# B&R Automation Studio project Assembly_and_ST (part 3)

#### Outfeed_Aborted.st
```iecst
ACTION Outfeed_Aborted:

	IF gSuperTrak.state.stateMachine.operationalState = ABORTED THEN
		//TODO: Insert Outfeed LED Light control

	ELSE
		//TODO: Insert Outfeed LED Light control
	END_IF;

	IF gSuperTrak.skill.Outfeed.state.stateMachine.stateTransition.reset THEN
		gSuperTrak.skill.Outfeed.state.stateMachine.operationalState := RESETTING;

	ELSIF gSuperTrak.skill.Outfeed.state.stateMachine.stateTransition.clear THEN
		gSuperTrak.skill.Outfeed.state.stateMachine.operationalState := CLEARING;

	END_IF;

END_ACTION
```

#### Outfeed_Stopped.st
```iecst
ACTION Outfeed_Stopped:

	IF gSuperTrak.skill.Outfeed.state.stateMachine.stateTransition.reset
	(*AND	NOT gbMessageSumAlarm*) THEN

		gSuperTrak.skill.Outfeed.state.stateMachine.operationalState := RESETTING;
	END_IF;

END_ACTION
```

#### Outfeed_Clearing.st
```iecst
ACTION Outfeed_Clearing:

	gSuperTrak.skill.Outfeed.state.stateMachine.stateTransition.clear := FALSE;

	gSuperTrak.skill.Outfeed.state.stateMachine.operationalState := STOPPED;

END_ACTION
```

#### Outfeed_Starting.st
```iecst
ACTION Outfeed_Starting:

	(* ************************************************************************** *)
	(* starting Outfeed skill *)
	IF NOT Outfeed_Full THEN
		gSuperTrak.skill.Outfeed.state.stateMachine.stateTransition.start := FALSE;
		gSuperTrak.skill.Outfeed.state.stateMachine.operationalState := RUNNING;
	END_IF;

END_ACTION
```

#### Outfeed_Completing.st
```iecst
ACTION Outfeed_Completing:
	gSuperTrak.skill.Outfeed.state.stateMachine.operationalState := COMPLETE;
END_ACTION
```

#### Outfeed_Complete.st
```iecst
ACTION Outfeed_Complete:

	Outfeed_Actuator_UP := FALSE;
	Outfeed_Actuator_DOWN := FALSE;
	Outfeed_Actuator_FRONT := FALSE;
	Outfeed_Actuator_BACK := FALSE;

	(* Skill stays in complete until trigger from MES *)
	IF gSuperTrak.skill.Outfeed.state.stateMachine.stateTransition.reset THEN
		gSuperTrak.skill.Outfeed.state.stateMachine.operationalState := RESETTING;
	END_IF;

END_ACTION
```

#### Outfeed_Holding.st
```iecst
ACTION Outfeed_Holding:

	gSuperTrak.skill.Outfeed.state.stateMachine.operationalState := HELD;

END_ACTION
```

#### Outfeed_Suspended.st
```iecst
ACTION Outfeed_Suspended:

	IF gSuperTrak.skill.Outfeed.state.stateMachine.stateTransition.unsuspend THEN
		gSuperTrak.skill.Outfeed.state.stateMachine.operationalState := UNSUSPENDING;
	END_IF;

END_ACTION
```

#### Outfeed_Unsuspending.st
```iecst
ACTION Outfeed_Unsuspending:

	gSuperTrak.skill.Outfeed.state.stateMachine.operationalState := RUNNING;

END_ACTION
```

#### Outfeed_Running.st
```iecst
ACTION Outfeed_Running:

	IF NOT Outfeed_Full AND Outfeed_Checked THEN
		(*Activate actuator movement up and wait until fully extended*)

		Outfeed_Actuator_UP := TRUE;

		Timer_Outfeed_UP(IN := TRUE, PT := T#10s);

		IF Timer_Outfeed_UP.Q THEN
			Outfeed_LED_Green := TRUE;
			Outfeed_LED_Red := FALSE;
			Outfeed_LED_Blue := FALSE;

			Outfeed_Actuator_FRONT := TRUE;
			Timer_Outfeed_FRONT(IN:= TRUE, PT:=T#5s);

			IF Timer_Outfeed_FRONT.Q THEN

				(*Actuator go down and then we get complete*)
				Outfeed_Actuator_UP := FALSE;
				Outfeed_Actuator_FRONT := FALSE;

				IF NOT Outfeed_Actuator_UP AND NOT Outfeed_Actuator_FRONT THEN
					Outfeed_Actuator_DOWN := TRUE;
					Outfeed_Actuator_BACK := TRUE;
				END_IF;

				Timer_Outfeed_DOWN(IN := Outfeed_Actuator_DOWN, PT := T#10s);
				Timer_Outfeed_BACK(IN := Outfeed_Actuator_BACK, PT := T#5s);

				IF Timer_Outfeed_DOWN.Q AND Timer_Outfeed_BACK.Q THEN
					Timer_Outfeed_DOWN(IN := FALSE);
					Timer_Outfeed_BACK(IN := FALSE);
					Timer_Outfeed_FRONT(IN := FALSE);
					Timer_Outfeed_UP (IN := FALSE);
					gSuperTrak.skill.Outfeed.state.stateMachine.operationalState := COMPLETING;
				END_IF;

			END_IF;

		END_IF;

	ELSIF NOT Outfeed_Checked THEN

		IF Outfeed_Full THEN
			Event_Code := 80;
			EventLog.Commands.WriteUserEvent := TRUE;

		ELSE
			Outfeed_Checked := TRUE;
		END_IF;

	END_IF;

END_ACTION
```

#### QACheck.st
```iecst
ACTION QACheck:
		(*************************************************************************************************)
		(*************************************************************************************************)
		(* State Machine *)
	CASE gSuperTrak.skill.QACheck.state.stateMachine.operationalState OF
		(*************************************************************************************************)
		(* RESETTING *)
		RESETTING:
			(*gSuperTrak.skill.QACheck.state.stateMachine.stateTransition.reset := FALSE;*)

			IF gSuperTrak.skill.QACheck.state.stateMachine.stateTransition.abort THEN
				gSuperTrak.skill.QACheck.state.stateMachine.operationalState := ABORTING;

			ELSIF gSuperTrak.skill.QACheck.state.stateMachine.stateTransition.stop THEN
				gSuperTrak.skill.QACheck.state.stateMachine.operationalState := STOPPING;

			ELSE
				QACheck_Resetting;

			END_IF;

		(*************************************************************************************************)
		(* IDLE *)
		IDLE:
			gSuperTrak.skill.QACheck.state.stateMachine.stateTransition.reset := FALSE;

			IF gSuperTrak.skill.QACheck.state.stateMachine.stateTransition.abort THEN
				gSuperTrak.skill.QACheck.state.stateMachine.operationalState := ABORTING;

			ELSIF gSuperTrak.skill.QACheck.state.stateMachine.stateTransition.stop THEN
				gSuperTrak.skill.QACheck.state.stateMachine.operationalState := STOPPING;

			ELSE
				QACheck_Idle;

			END_IF;

		(*************************************************************************************************)
		(* STARTING *)
		STARTING:
//			gSuperTrak.skill.QACheck.state.stateMachine.stateTransition.start := FALSE;

			IF gSuperTrak.skill.QACheck.state.stateMachine.stateTransition.abort THEN
				gSuperTrak.skill.QACheck.state.stateMachine.operationalState := ABORTING;

			ELSIF gSuperTrak.skill.QACheck.state.stateMachine.stateTransition.stop THEN
				gSuperTrak.skill.QACheck.state.stateMachine.operationalState := STOPPING;

			ELSE
				QACheck_Starting;

			END_IF;

		(*************************************************************************************************)
		(* RUNNING *)
		RUNNING:

			gSuperTrak.skill.QACheck.state.stateMachine.stateTransition.start := FALSE;

			IF gSuperTrak.skill.QACheck.state.stateMachine.stateTransition.abort THEN
				gSuperTrak.skill.QACheck.state.stateMachine.operationalState := ABORTING;

			ELSIF gSuperTrak.skill.QACheck.state.stateMachine.stateTransition.stop THEN
				gSuperTrak.skill.QACheck.state.stateMachine.operationalState := STOPPING;

			ELSIF gSuperTrak.skill.QACheck.state.stateMachine.stateTransition.hold THEN

				//				gSuperTrak.skill.QACheck.state.stateMachine.operationalState := HOLDING;

			ELSIF gSuperTrak.skill.QACheck.state.stateMachine.stateTransition.suspend THEN

				//				gSuperTrak.skill.QACheck.state.stateMachine.operationalState := SUSPENDING;

			ELSIF gSuperTrak.skill.QACheck.state.stateMachine.stateTransition.pause THEN

				//				gSuperTrak.skill.QACheck.state.stateMachine.operationalState := PAUSING;

			ELSE
				QACheck_Running;

			END_IF;

		(*************************************************************************************************)
		(* PAUSING *)
		PAUSING:
			(*gSuperTrak.skill.QACheck.state.stateMachine.stateTransition.pause := FALSE;*)

			IF gSuperTrak.skill.QACheck.state.stateMachine.stateTransition.abort THEN
				gSuperTrak.skill.QACheck.state.stateMachine.operationalState := ABORTING;

			ELSIF gSuperTrak.skill.QACheck.state.stateMachine.stateTransition.stop THEN
				gSuperTrak.skill.QACheck.state.stateMachine.operationalState := STOPPING;

			ELSIF gSuperTrak.skill.QACheck.state.stateMachine.stateTransition.hold THEN

				//				gSuperTrak.skill.QACheck.state.stateMachine.operationalState := HOLDING;

			ELSIF gSuperTrak.skill.QACheck.state.stateMachine.stateTransition.suspend THEN

				//				gSuperTrak.skill.QACheck.state.stateMachine.operationalState := SUSPENDING;

			ELSE
				QACheck_Pausing;
			END_IF;

		(*************************************************************************************************)
		(* PAUSED *)
		PAUSED:

			gSuperTrak.skill.QACheck.state.stateMachine.stateTransition.pause := FALSE;

			IF gSuperTrak.skill.QACheck.state.stateMachine.stateTransition.abort THEN
				gSuperTrak.skill.QACheck.state.stateMachine.operationalState := ABORTING;

			ELSIF gSuperTrak.skill.QACheck.state.stateMachine.stateTransition.stop THEN
				gSuperTrak.skill.QACheck.state.stateMachine.operationalState := STOPPING;

			ELSIF gSuperTrak.skill.QACheck.state.stateMachine.stateTransition.hold THEN

				//				gSuperTrak.skill.QACheck.state.stateMachine.operationalState := HOLDING;

			ELSIF gSuperTrak.skill.QACheck.state.stateMachine.stateTransition.suspend THEN

				//				gSuperTrak.skill.QACheck.state.stateMachine.operationalState := SUSPENDING;

			ELSE
				QACheck_Paused;

			END_IF;

		(*************************************************************************************************)
		(* SUSPENDING *)
		SUSPENDING:
			(*gSuperTrak.skill.QACheck.state.stateMachine.stateTransition.suspend := FALSE;*)

			IF gSuperTrak.skill.QACheck.state.stateMachine.stateTransition.abort THEN
				gSuperTrak.skill.QACheck.state.stateMachine.operationalState := ABORTING;

			ELSIF gSuperTrak.skill.QACheck.state.stateMachine.stateTransition.stop THEN
				gSuperTrak.skill.QACheck.state.stateMachine.operationalState := STOPPING;

			ELSIF gSuperTrak.skill.QACheck.state.stateMachine.stateTransition.hold THEN

				//				gSuperTrak.skill.QACheck.state.stateMachine.operationalState := HOLDING;

			ELSE
				QACheck_Suspending;

			END_IF;

		(*************************************************************************************************)
		(* SUSPENDED *)
		SUSPENDED:

			gSuperTrak.skill.QACheck.state.stateMachine.stateTransition.suspend := FALSE;

			IF gSuperTrak.skill.QACheck.state.stateMachine.stateTransition.abort THEN
				gSuperTrak.skill.QACheck.state.stateMachine.operationalState := ABORTING;

			ELSIF gSuperTrak.skill.QACheck.state.stateMachine.stateTransition.stop THEN
				gSuperTrak.skill.QACheck.state.stateMachine.operationalState := STOPPING;

			ELSIF gSuperTrak.skill.QACheck.state.stateMachine.stateTransition.hold THEN

				//				gSuperTrak.skill.QACheck.state.stateMachine.operationalState := HOLDING;

			ELSE
				QACheck_Suspended;

			END_IF;

		(*************************************************************************************************)
		(* UNSUSPENDING *)
		UNSUSPENDING:
			gSuperTrak.skill.QACheck.state.stateMachine.stateTransition.unsuspend := FALSE;

			IF gSuperTrak.skill.QACheck.state.stateMachine.stateTransition.abort THEN
				gSuperTrak.skill.QACheck.state.stateMachine.operationalState := ABORTING;

			ELSIF gSuperTrak.skill.QACheck.state.stateMachine.stateTransition.stop THEN
				gSuperTrak.skill.QACheck.state.stateMachine.operationalState := STOPPING;

			ELSIF gSuperTrak.skill.QACheck.state.stateMachine.stateTransition.hold THEN

				//				gSuperTrak.skill.QACheck.state.stateMachine.operationalState := HOLDING;

			ELSE
				QACheck_Unsuspending;

			END_IF;

		(*************************************************************************************************)
		(* HOLDING *)
		HOLDING:
			(*gSuperTrak.skill.QACheck.state.stateMachine.stateTransition.hold := FALSE;*)

			IF gSuperTrak.skill.QACheck.state.stateMachine.stateTransition.abort THEN
				gSuperTrak.skill.QACheck.state.stateMachine.operationalState := ABORTING;

			ELSIF gSuperTrak.skill.QACheck.state.stateMachine.stateTransition.stop THEN
				gSuperTrak.skill.QACheck.state.stateMachine.operationalState := STOPPING;

			ELSE
				QACheck_Holding;

			END_IF;

		(*************************************************************************************************)
		(* HELD *)
		HELD:

			gSuperTrak.skill.QACheck.state.stateMachine.stateTransition.hold := FALSE;

			IF gSuperTrak.skill.QACheck.state.stateMachine.stateTransition.abort THEN
				gSuperTrak.skill.QACheck.state.stateMachine.operationalState := ABORTING;

			ELSIF gSuperTrak.skill.QACheck.state.stateMachine.stateTransition.stop THEN
				gSuperTrak.skill.QACheck.state.stateMachine.operationalState := STOPPING;

			ELSE
				QACheck_Held;

			END_IF;

		(*************************************************************************************************)
		(* UNHOLDING *)
		UNHOLDING:
			gSuperTrak.skill.QACheck.state.stateMachine.stateTransition.unhold := FALSE;

			IF gSuperTrak.skill.QACheck.state.stateMachine.stateTransition.abort THEN
				gSuperTrak.skill.QACheck.state.stateMachine.operationalState := ABORTING;

			ELSIF gSuperTrak.skill.QACheck.state.stateMachine.stateTransition.stop THEN
				gSuperTrak.skill.QACheck.state.stateMachine.operationalState := STOPPING;

			ELSE
				QACheck_Unholding;

			END_IF;

		(*************************************************************************************************)
		(* COMPLETING *)
		COMPLETING:

			IF gSuperTrak.skill.QACheck.state.stateMachine.stateTransition.abort THEN
				gSuperTrak.skill.QACheck.state.stateMachine.operationalState := ABORTING;

			ELSIF gSuperTrak.skill.QACheck.state.stateMachine.stateTransition.stop THEN
				gSuperTrak.skill.QACheck.state.stateMachine.operationalState := STOPPING;

			ELSE
				QACheck_Completing;

			END_IF;

		(*************************************************************************************************)
		(* COMPLETE *)
		COMPLETE:

			IF gSuperTrak.skill.QACheck.state.stateMachine.stateTransition.abort THEN
				gSuperTrak.skill.QACheck.state.stateMachine.operationalState := ABORTING;

			ELSIF gSuperTrak.skill.QACheck.state.stateMachine.stateTransition.stop THEN
				gSuperTrak.skill.QACheck.state.stateMachine.operationalState := STOPPING;

			ELSE
				QACheck_Complete;

			END_IF;

		(*************************************************************************************************)
		(* STOPPING *)
		STOPPING:
//			gSuperTrak.skill.QACheck.state.stateMachine.stateTransition.stop := FALSE;

			IF gSuperTrak.skill.QACheck.state.stateMachine.stateTransition.abort THEN
				gSuperTrak.skill.QACheck.state.stateMachine.operationalState := ABORTING;

			ELSE
				QACheck_Stopping;

			END_IF;

		(*************************************************************************************************)
		(* STOPPED *)
		STOPPED:

			gSuperTrak.skill.QACheck.state.stateMachine.stateTransition.stop := FALSE;

			IF gSuperTrak.skill.QACheck.state.stateMachine.stateTransition.abort THEN
				gSuperTrak.skill.QACheck.state.stateMachine.operationalState := ABORTING;

			ELSE
				QACheck_Stopped;

			END_IF;

		(*************************************************************************************************)
		(* ABORTING *)
		ABORTING:
			(*gSuperTrak.skill.QACheck.state.stateMachine.stateTransition.abort := FALSE;*)

			QACheck_Aborting;

		(*************************************************************************************************)
		(* ABORTED *)
		ABORTED:

			gSuperTrak.skill.QACheck.state.stateMachine.stateTransition.abort := FALSE;

			QACheck_Aborted;

		(*************************************************************************************************)
		(* CLEARING *)
		CLEARING:
			gSuperTrak.skill.QACheck.state.stateMachine.stateTransition.clear := FALSE;

			QACheck_Clearing;

			(*************************************************************************************************)
			(* ELSE *)
		ELSE;

	END_CASE;
END_ACTION
```

#### QACheck_Aborting.st
```iecst
ACTION QACheck_Aborting:

//	IF NOT Transition_From_Stopped AND gSuperTrak.state.stateMachine.operationalState <> ABORTING THEN
//		Event_Code := 77;
//		EventLog.Commands.WriteUserEvent := TRUE;
//	END_IF;
//

	//Not knowing if any trigger was set to true before the abort we make sure every one of them is false before going to aborted
	gSuperTrak.skill.QACheck.state.stateMachine.stateTransition.abort 		:= FALSE;
	gSuperTrak.skill.QACheck.state.stateMachine.stateTransition.clear 		:= FALSE;
	gSuperTrak.skill.QACheck.state.stateMachine.stateTransition.hold 		:= FALSE;
	gSuperTrak.skill.QACheck.state.stateMachine.stateTransition.pause 		:= FALSE;
	gSuperTrak.skill.QACheck.state.stateMachine.stateTransition.reset 		:= FALSE;
	gSuperTrak.skill.QACheck.state.stateMachine.stateTransition.resume 		:= FALSE;
	gSuperTrak.skill.QACheck.state.stateMachine.stateTransition.start 		:= FALSE;
	gSuperTrak.skill.QACheck.state.stateMachine.stateTransition.stop 		:= FALSE;
	gSuperTrak.skill.QACheck.state.stateMachine.stateTransition.suspend 	:= FALSE;
	gSuperTrak.skill.QACheck.state.stateMachine.stateTransition.unhold 		:= FALSE;
	gSuperTrak.skill.QACheck.state.stateMachine.stateTransition.unsuspend 	:= FALSE;

	LED_Red   := TRUE;
	LED_Green := FALSE;
	LED_Blue  := FALSE;
	QA_Actuator_UP := FALSE;

	QA_Actuator_DOWN := FALSE;

	Skills_Aborted := Skills_Aborted + 1;
	gSuperTrak.skill.QACheck.state.stateMachine.operationalState := ABORTED;

END_ACTION
```

#### QACheck_Aborted.st
```iecst
ACTION QACheck_Aborted:

	IF gSuperTrak.state.stateMachine.operationalState = ABORTED THEN
		LED_Blue := TRUE;
		LED_Green := FALSE;
		LED_Red := FALSE;

	ELSE
		LED_Blue := FALSE;
		LED_Green := FALSE;
		LED_Red := TRUE;
	END_IF;

	IF gSuperTrak.skill.QACheck.state.stateMachine.stateTransition.reset THEN
		gSuperTrak.skill.QACheck.state.stateMachine.operationalState := RESETTING;

	ELSIF gSuperTrak.skill.QACheck.state.stateMachine.stateTransition.clear THEN
		gSuperTrak.skill.QACheck.state.stateMachine.operationalState := CLEARING;

	END_IF;

END_ACTION
```

#### QACheck_Clearing.st
```iecst
ACTION QACheck_Clearing:

	gSuperTrak.skill.QACheck.state.stateMachine.stateTransition.clear := FALSE;

	gSuperTrak.skill.QACheck.state.stateMachine.operationalState := STOPPED;

END_ACTION
```

#### QACheck_Idle.st
```iecst
ACTION QACheck_Idle:

	LED_Green := FALSE;
	LED_Red := FALSE;
	LED_Blue := TRUE;

	IF gSuperTrak.skill.QACheck.state.stateMachine.stateTransition.start THEN

		gSuperTrak.skill.QACheck.state.stateMachine.operationalState := STARTING;

	END_IF

	QA_Actuator_UP := FALSE;
	QA_Actuator_DOWN := FALSE;

END_ACTION
```

#### QACheck_Starting.st
```iecst
ACTION QACheck_Starting:

	(* ************************************************************************** *)
	(* starting QACheck skill *)
	gSuperTrak.skill.QACheck.state.stateMachine.stateTransition.start := FALSE;
	gSuperTrak.skill.QACheck.state.stateMachine.operationalState := RUNNING;

END_ACTION
```

#### QACheck_Completing.st
```iecst
ACTION QACheck_Completing:

	(* Alarms Handling?? *)

	(*Actuator go down and then we get complete*)
	QA_Actuator_UP := FALSE;
	LED_Green := FALSE;
	LED_Red := TRUE;
	LED_Blue := FALSE;
	Timer_Enable_Barrier(IN := LED_Red, PT := T#0.5s);

	IF Timer_Enable_Barrier.Q THEN
		Disable_Light_Barrier := FALSE;
	END_IF;

	IF NOT QA_Actuator_UP THEN
		QA_Actuator_DOWN := TRUE;
	END_IF;

	Timer_Actuator_DOWN(IN := QA_Actuator_DOWN, PT := T#8s);

	IF Timer_Actuator_DOWN.Q AND NOT Disable_Light_Barrier THEN
		gSuperTrak.skill.QACheck.state.stateMachine.operationalState := COMPLETE;
		Timer_Actuator_DOWN(IN := FALSE);
	END_IF;

END_ACTION
```

#### QACheck_Complete.st
```iecst
ACTION QACheck_Complete:
	(* Skill stays in complete until trigger from MES *)
	IF gSuperTrak.skill.QACheck.state.stateMachine.stateTransition.reset THEN
		gSuperTrak.skill.QACheck.state.stateMachine.operationalState := RESETTING;
	END_IF;

	Timer_Enable_Barrier(IN := FALSE);
	QA_Actuator_UP := FALSE;
	QA_Actuator_DOWN := FALSE;

END_ACTION
```

#### QACheck_Running.st
```iecst
ACTION QACheck_Running:
	(*Activate actuator movement up and wait until fully extended*)

	Timer_Actuator_UP(IN := QA_Actuator_UP, PT := T#8s);
	QA_Actuator_UP := TRUE;

	IF Timer_Actuator_UP.Q THEN
		LED_Green := TRUE;
		LED_Red := FALSE;
		LED_Blue := FALSE;
		Disable_Light_Barrier := TRUE;
	END_IF;

	IF QA_finished THEN
		QA_finished := FALSE;
		QA_Actuator_UP := FALSE;
		Timer_Actuator_UP(IN := FALSE);
		gSuperTrak.skill.QACheck.state.stateMachine.operationalState := COMPLETING;
	END_IF;

END_ACTION
```

### UsrEventHandling.typ
```iecst
(*******************************************************************
 * Local data types of program EventLog
 ********************************************************************)

TYPE
	EventLog_typ : 	STRUCT  (*Event handling.*)
		Commands : EventLog_Commands_typ; (*Event handling user commands.*)
		Data : EventLog_Data_typ; (*Event handling data for state machine.*)
		Event : EventLog_Event_typ; (*Event handling event description.*)
		FunctionBlocks : EventLog_FunctionBlocks_typ; (*Event handling used function blocks.*)
	END_STRUCT;
	EventLog_Data_typ : 	STRUCT
		Step : EventLogSteps; (*Current step. STEP_ERROR must be manually reset (STEP_WAIT_FOR_INPUT).*)
		Ident : ArEventLogIdentType; (*Ident of the logbook "UsrEvLog".*)
		StatusID : DINT; (*Status information for STEP_ERROR.*)
		GetIdentOkNextStep : EventLogSteps; (*Internal helper for state machine.*)
		GetIdentFailNextStep : EventLogSteps; (*Internal helper for state machine.*)
	END_STRUCT;
	EventLog_Event_typ : 	STRUCT
		Severity : USINT; (*Severity of the last event (read).*)
		Customer : BOOL; (*Customer bit of the last event (read).*)
		Facility : UINT; (*Facility of the last event (read).*)
		Code : UINT; (*Code of the last event (read).*)
		EventID : DINT; (*EventID for write event (write - is not set by reading an event).*)
		ErrorNumber : UDINT; (*Error number of the event - set when the read event is no event id event (read).*)
		EnteredBy : STRING[36]; (*User/object identification (read/write - optional).*)
		OriginID : ArEventLogRecordIDType; (*Record id of the origin record (read/write - optional).*)
		RecordID : ArEventLogRecordIDType; (*Record id of the event to read (read - set automatically).*)
		TimeStamp : ArEventLogTimeStampType;
		AdditionalDataSize : UDINT; (*Size of the additional data (read/write - optional)*)
		AdditionalDataFormat : USINT; (*Format of the additional data (read/write)*)
		AdditionalData : STRING[255]; (*Additional data (read/write)*)
	END_STRUCT;
	EventLog_FunctionBlocks_typ : 	STRUCT
		ArEventLogCreate_0 : ArEventLogCreate;
		ArEventLogDelete_0 : ArEventLogDelete;
		ArEventLogGetIdent_0 : ArEventLogGetIdent;
		ArEventLogGetLatestRecordID_0 : ArEventLogGetLatestRecordID;
		ArEventLogGetPreviousRecordID_0 : ArEventLogGetPreviousRecordID;
		ArEventLogWrite_0 : ArEventLogWrite;
		ArEventLogRead_0 : ArEventLogRead;
		ArEventLogReadErrorNumber_0 : ArEventLogReadErrorNumber;
		ArEventLogReadAddData_0 : ArEventLogReadAddData;
		ArEventLogReadObjectID_0 : ArEventLogReadObjectID;
	END_STRUCT;
	EventLogSteps :
		(
		STEP_WAIT_FOR_INPUT := 0,
		STEP_CREATE_LOGBOOK := 1,
		STEP_DELETE_LOGBOOK := 2,
		STEP_GET_LOGBOOK_IDENT := 3,
		STEP_WRITE_EVENT := 4,
		STEP_READ_EVENT := 5,
		STEP_READ_ERROR_NUMBER := 6,
		STEP_READ_ADDITIONAL_DATA := 7,
		STEP_READ_OBJECT_ID := 8,
		STEP_GET_LATEST_RECORD_ID := 9,
		STEP_GET_PREVIOUS_RECORD_ID := 10,
		STEP_ERROR := 255
		);
END_TYPE

(*
Copyright ATS Automation Tooling Systems, Inc. 2015-2016
All rights reserved.
*)
(********************************************************************
 * COPYRIGHT --
 ********************************************************************
 * File: Global.typ
 * Author: VM_User
 * Created: 14. März 2014
 ********************************************************************
 * Global data types of project T1
 ********************************************************************)
(***********************************************************************)
(*Variables for Event logger control and definition*)
(**********************************************************************)

TYPE
	EventLog_Commands_typ : 	STRUCT
		CreateUserLog : BOOL; (*Creates the user logbook "UsrEvLog" in USERROM.*)
		DeleteUserLog : BOOL; (*Deletes the user logbook "UsrEvLog".*)
		WriteUserEvent : BOOL; (*Writes a user event into the user logbook "UsrEvLog". *)
		ReadLatestEvent : BOOL; (*Reads the latest event of the user logbook "UsrEvLog".*)
		ReadPreviousEvent : BOOL; (*Reads the previous event (of the given record id) of the user logbook "UserEvLog".*)
	END_STRUCT;
	Event_Codes_Typ : 	STRUCT
		Severity_Code : USINT;
		Facility_Code : USINT;
		Code_Value : USINT;
		ID : DINT;
		Event_Message : STRING[256]; (*Message for the event generated*)
	END_STRUCT;
END_TYPE
```

### UsrEventHandling.var
```iecst
(* ============================================================
Variable for known events definition
   ============================================================ *)
VAR
	Events : ARRAY[0..250] OF Event_Codes_Typ;
	Event_Code : UINT;
END_VAR
(*******************************************************************
 * Variables of program EventLog
 ********************************************************************)
VAR
	EventLog : EventLog_typ; (*Event handling.*)
END_VAR
(*=============================================================*)
(*Variables for info events writing control*)
(*=============================================================*)
VAR
	Write_Info : BOOL;
	ST_Last_Info_Written : UINT;
	Assembly_Last_Info_Written : UINT;
	General_Last_Info_Written : UINT;
	Last_Event_Written : UINT;
	Set_Info_Messages : BOOL;
	Restart_Status : UINT;
	Initialization : BOOL;
END_VAR
(*=============================================================*)
(*Flags for new events *)
(*=============================================================*)
VAR
	Info_Event : BOOL;
	New_Event : BOOL;
END_VAR
(********************************************************************************************)
(* Variables for Error Detection *)
(********************************************************************************************)
VAR
	SumCritical : BOOL;
END_VAR
```

### Program Logical/Events_handling/AlarmHandling

#### Variables.var
```iecst
VAR
	i : USINT;
	iEvent : USINT := 0;
END_VAR
(********************************************************************************************)
(* Variables for Service Stations *)
(********************************************************************************************)
VAR
END_VAR
```

#### Main.st
```iecst
PROGRAM _INIT
	(*Initial definiton of all the messages that could possibly be used during the execution*)
	ST_Events_Data;
	Assembly_Events_Data;
	General_Events_Data;

	(*Flag for the user to select whether or not the info messages of the actual state of the state machines will be shown*)
	//By default is false taking into account that if not this could generate execesive information in the logger
	Set_Info_Messages := FALSE;
	SumCritical := FALSE;

	Initialization := TRUE;

END_PROGRAM

PROGRAM _CYCLIC
	ComauerrorHandler;
	STerrorHandler;
	RefillEvent;
	ErrorSum;
	(* Error Reset *)

	IF gSuperTrak.state.errorAcknowledge AND SumCritical THEN

		IF Last_Event_Written = 200  AND NOT Initialization THEN
			Event_Code := 201;
			EventLog.Commands.WriteUserEvent := TRUE;

			Restart_Status := SYSreset(1, 1); (* perform WARMSTART *)

			IF Restart_Status <> 0 THEN (* check status value *)
				Event_Code := 202;
				EventLog.Commands.WriteUserEvent := TRUE;
			END_IF;

		END_IF;

		Event_Code := 249;
		EventLog.Commands.WriteUserEvent := TRUE;
		Initialization := FALSE;

		gSuperTrak.state.errorAcknowledge := FALSE;
		SumCritical := FALSE;

	END_IF;

	IF gAssemblyModule.state.errorAcknowledge AND SumCritical THEN

		IF Last_Event_Written = 200  AND NOT Initialization THEN
			Event_Code := 201;
			EventLog.Commands.WriteUserEvent := TRUE;

			Restart_Status := SYSreset(1, 1); (* perform WARMSTART *)

			IF Restart_Status <> 0 THEN (* check status value *)
				Event_Code := 202;
				EventLog.Commands.WriteUserEvent := TRUE;
			END_IF;

		END_IF;

		Event_Code := 249;
		EventLog.Commands.WriteUserEvent := TRUE;

		gAssemblyModule.state.errorAcknowledge := FALSE;
		SumCritical := FALSE;

	END_IF;

	StateInfo;
	ServiceStations;
	Assembly_WarningHandler;

	(* Call to the skills responsible of the critical errors detection and duplicate messages management*)
	IF New_Event THEN
		InfoHistory;
	END_IF;

END_PROGRAM
```

#### ComauErrorHandler.st
```iecst
ACTION ComauerrorHandler:

	IF Event_Code = 101 THEN

		Mp_Comau.ErrorReset := TRUE;

		Plastic_Cup_Supply_Position[0] := PLASTIC_CUP_INIT_POSITION [0];
		Plastic_Cup_Supply_Position[1] := PLASTIC_CUP_INIT_POSITION [1];
		Plastic_Cup_Supply_Position[2] := PLASTIC_CUP_INIT_POSITION [2];

		Plastic_Cup_Supply_Above_Pos[0] := PLASTIC_CUP_INIT_POSITION [0];
		Plastic_Cup_Supply_Above_Pos[1] := PLASTIC_CUP_INIT_POSITION [1];
		Plastic_Cup_Supply_Above_Pos[2] := PLASTIC_CUP_INIT_POSITION [2] + 60;

		x_counter_plastic := 0;
		y_counter_plastic := 0;

		Paper_Cup_Supply_Position[0] := PAPER_CUP_INIT_POSITION [0];
		Paper_Cup_Supply_Position[1] := PAPER_CUP_INIT_POSITION [1];
		Paper_Cup_Supply_Position[2] := PAPER_CUP_INIT_POSITION [2];

		Paper_Cup_Supply_Above_Pos[0] := PAPER_CUP_INIT_POSITION [0];
		Paper_Cup_Supply_Above_Pos[1] := PAPER_CUP_INIT_POSITION [1];
		Paper_Cup_Supply_Above_Pos[2] := PAPER_CUP_INIT_POSITION [2] + 60;

		x_counter_plastic := 0;
		y_counter_plastic := 0;

		IF NOT Mp_Comau.Error THEN
			Mp_Comau.ErrorReset := FALSE;
		END_IF;

	END_IF;

	IF Event_Code = 102 THEN  //Error in imput parameter paper cup
		gAssemblyModule.skill.provideCup.inputParameters.cupType :=0;
	END_IF;

	IF Event_Code = 131 //Error In Homing Procedure
		OR Event_Code = 100 THEN //Clearing Timeout

		Mp_Comau.ErrorReset := TRUE;
		Mp_Comau.Home := FALSE;
		HomeRobot := FALSE;

		IF NOT Mp_Comau.Error THEN
			Mp_Comau.ErrorReset := FALSE;
		END_IF;

	END_IF;

END_ACTION
```

#### STErrorHandler.st
```iecst
ACTION STerrorHandler:

	IF StControl_0.Error THEN
		Event_Code := 1;
		EventLog.Commands.WriteUserEvent := TRUE;
	END_IF;

END_ACTION
```

#### ErrorAcknowledgement.st - not listed in the package file held
```iecst
ACTION ErrorAcknowledgement:
	(* Error Reset *)
	IF gSuperTrak.state.errorAcknowledge AND SumCritical THEN

		Event_Code := 249;
		EventLog.Commands.WriteUserEvent := TRUE;

		gSuperTrak.state.errorAcknowledge := FALSE;
		SumCritical := FALSE;

	END_IF;

	IF gAssemblyModule.state.errorAcknowledge AND SumCritical THEN

		Event_Code := 249;
		EventLog.Commands.WriteUserEvent := TRUE;

		gAssemblyModule.state.errorAcknowledge := FALSE;
		SumCritical := FALSE;
	END_IF;

END_ACTION
```

#### InfoHistory.st
```iecst
ACTION InfoHistory:

	EventLog.Commands.ReadLatestEvent := TRUE;

	IF EventLog.FunctionBlocks.ArEventLogReadObjectID_0.Done THEN

		IF Info_Event THEN

			IF EventLog.Event.Code < 100 THEN
				ST_Last_Info_Written := EventLog.Event.Code;

			ELSIF EventLog.Event.Code < 200 THEN
				Assembly_Last_Info_Written := EventLog.Event.Code;

			ELSE
				General_Last_Info_Written := EventLog.Event.Code;
			END_IF;

		ELSE

			Last_Event_Written := EventLog.Event.Code;

		END_IF;

		New_Event := FALSE;

	END_IF;

END_ACTION
```

#### Refill_Event.st
```iecst
ACTION RefillEvent:

	//If a refill event is reached the module will be held, as well as the skill that detected the empty storage
	IF Event_Code = 130 THEN

		Assem_IgnoreSafetySensors := TRUE;

		IF Assem_PaperRemaining = 0 THEN
			Paper_RefillDone := FALSE;
		END_IF;

		IF Assem_PlasticRemaining = 0 THEN
			Plastic_RefillDone := FALSE;
		END_IF;

		IF gAssemblyModule.skill.provideCup.state.stateMachine.operationalState = RUNNING THEN

			gAssemblyModule.skill.provideCup.state.stateMachine.stateTransition.hold := TRUE;

		END_IF;

		IF gAssemblyModule.skill.providePellet.state.stateMachine.operationalState = RUNNING THEN

			gAssemblyModule.skill.providePellet.state.stateMachine.stateTransition.hold := TRUE;

		END_IF;

		gAssemblyModule.state.stateMachine.stateTransition.hold := TRUE;

	END_IF;

	//If a refill event is reached the module will be held, as well as the skill that detected the empty storage
	IF Event_Code = 133 THEN

		IF gAssemblyModule.skill.provideCup.state.stateMachine.operationalState = HELD THEN

			gAssemblyModule.skill.provideCup.state.stateMachine.stateTransition.unhold := TRUE;

		END_IF;

		IF gAssemblyModule.skill.providePellet.state.stateMachine.operationalState = HELD THEN

			gAssemblyModule.skill.providePellet.state.stateMachine.stateTransition.unhold := TRUE;

		END_IF;

		gAssemblyModule.state.stateMachine.stateTransition.unhold := TRUE;

	END_IF;

	IF Last_Event_Written = 133 THEN
		Event_Code := 141;
		EventLog.Commands.WriteUserEvent := TRUE;
	END_IF;

	IF gAssemblyModule.state.stateMachine.operationalState = RUNNING THEN

		//Assem_IgnoreSafetySensors := FALSE;
		gAssemblyModule.state.stateMachine.stateTransition.unhold := FALSE;

	END_IF;

	//When the refill has been completed the three refill variables will be true and the pellets will be
	//detected by the light barrier
	IF Plastic_RefillDone AND Paper_RefillDone AND Assem_PelletPresent THEN
		Refill_Done := TRUE;
	END_IF;

END_ACTION
```

#### Demo_Mode.st - not listed in the package file held
```iecst
ACTION Demo_Mode:
//Mode where the whole process can be simulated wothout needing an MES execution.
//Only SuperTrak is controlled and the modules interaction is faked using timers for a realistic execution.

	IF gSuperTrak.state.stateMachine.operationalState = ABORTED
		AND SumCritical = FALSE THEN

		gSuperTrak.state.stateMachine.stateTransition.clear := TRUE;

	END_IF;

	IF gSuperTrak.state.stateMachine.operationalState = STOPPED THEN

		gSuperTrak.state.stateMachine.stateTransition.reset := TRUE;

	END_IF;

	IF gSuperTrak.state.stateMachine.operationalState = IDLE THEN

		gSuperTrak.state.stateMachine.stateTransition.start := TRUE;

	END_IF;

	IF  gSuperTrak.state.stateMachine.operationalState = RUNNING AND
		Place_Order AND (ID = 0 OR ID = -1) THEN

		//Call skill checkParking to retrieve shuttleID

		gSuperTrak.skill.checkParking.state.stateMachine.stateTransition.start := TRUE;

		//When skill is finished store the ID in a variable
		IF gSuperTrak.skill.checkParking.state.stateMachine.operationalState = COMPLETE THEN

			ID := gSuperTrak.skill.checkParking.outputParameters.shuttleId;
			gSuperTrak.skill.checkParking.state.stateMachine.stateTransition.reset := TRUE;

		END_IF;

	END_IF;

	//checkParking returns -1 if there is no shuttle there at the station
	IF ID <> -1 AND ID <> 0 AND StTargetExt_[1].PalletPresent THEN

		Place_Order := FALSE;
		ID := 0;
		TargetControlParameters[1].AdvancedReleaseConfig.DestinationTarget := 2;
		StTargetExt_[1].ReleaseToTarget := TRUE;

		IF EDGENEG(StTargetExt_[1].PalletPresent) THEN

			StTargetExt_[1].ReleaseToTarget := FALSE;

		END_IF;

	END_IF;

	//Assembly Module
	IF StTargetExt_[2].PalletPresent THEN

		TON_Release_Target_2 (IN := TRUE, PT := T#5s);

		IF TON_Release_Target_2.Q THEN

			StTargetExt_[2].ReleaseToTarget := TRUE;

		END_IF;

	END_IF;

	IF EDGENEG(StTargetExt_[2].PalletPresent) THEN

		StTargetExt_[2].ReleaseToTarget := FALSE;
		TON_Release_Target_2 (IN := FALSE);

	END_IF;

	//SeedSupply Module
	IF StTargetExt_[3].PalletPresent THEN

		TON_Release_Target_3 (IN := TRUE, PT := T#12s);

		IF TON_Release_Target_3.Q THEN

			IF StTargetExt_[1].PalletPresent THEN
				Get_away := TRUE;
			END_IF;

			StTargetExt_[3].ReleaseToTarget := TRUE;
			TON_Check_Parking (IN := TRUE, PT := T#3.5s);

		END_IF;

	END_IF;

	IF EDGENEG(StTargetExt_[3].PalletPresent) THEN

		StTargetExt_[3].ReleaseToTarget := FALSE;
		TON_Release_Target_3 (IN := FALSE);

	END_IF;

	IF StTargetExt_[1].PalletPresent AND NOT StTargetExt_[1].ReleaseToTarget
		AND NOT TON_Check_Parking.Q AND Get_away THEN

		TargetControlParameters[1].AdvancedReleaseConfig.DestinationTarget := 8;
		TargetControlParameters[1].AdvancedReleaseConfig.MoveConfigIdx := 2;
		StTargetExt_[1].ReleaseToTarget := TRUE;

	END_IF;

	IF TON_Check_Parking.Q THEN

		Get_away := FALSE;
		TON_Check_Parking (IN := FALSE);
		TargetControlParameters[1].AdvancedReleaseConfig.DestinationTarget := 2;
		TargetControlParameters[1].AdvancedReleaseConfig.MoveConfigIdx := 1;

	END_IF;

	IF EDGENEG(StTargetExt_[1].PalletPresent) THEN

		StTargetExt_[1].ReleaseToTarget := FALSE;

	END_IF;

	//QA Station
	IF StTargetExt_[4].PalletPresent THEN

		IF gSuperTrak.skill.QACheck.state.stateMachine.operationalState = IDLE THEN

			gSuperTrak.skill.QACheck.state.stateMachine.stateTransition.start := TRUE;

		ELSE

			gSuperTrak.skill.QACheck.state.stateMachine.stateTransition.start := FALSE;

		END_IF;

		IF gSuperTrak.skill.QACheck.state.stateMachine.operationalState = COMPLETE THEN

			gSuperTrak.skill.QACheck.state.stateMachine.stateTransition.reset := TRUE;
			StTargetExt_[4].ReleaseToTarget := TRUE;

		END_IF;

	END_IF;

	IF EDGENEG(StTargetExt_[4].PalletPresent) THEN

		StTargetExt_[4].ReleaseToTarget := FALSE;

	END_IF;

	//Sealing Module
	IF StTargetExt_[5].PalletPresent THEN

		TON_Release_Target_5 (IN := TRUE, PT := T#15s);

		IF TON_Release_Target_5.Q THEN

			StTargetExt_[5].ReleaseToTarget := TRUE;

		END_IF;

	END_IF;

	IF EDGENEG(StTargetExt_[5].PalletPresent) THEN

		StTargetExt_[5].ReleaseToTarget := FALSE;
		TON_Release_Target_5 (IN := FALSE);

	END_IF;

	//Labeling Module
	IF StTargetExt_[6].PalletPresent THEN

		TON_Release_Target_6 (IN := TRUE, PT := T#1s);

		IF TON_Release_Target_6.Q THEN

			StTargetExt_[6].ReleaseToTarget := TRUE;

		END_IF;

	END_IF;

	IF EDGENEG(StTargetExt_[6].PalletPresent) THEN

		StTargetExt_[6].ReleaseToTarget := FALSE;
		TON_Release_Target_6 (IN := FALSE);

	END_IF;

	//Outfeed Station
	IF StTargetExt_[7].PalletPresent THEN

		IF gSuperTrak.skill.Outfeed.state.stateMachine.operationalState = IDLE THEN

			gSuperTrak.skill.Outfeed.state.stateMachine.stateTransition.start := TRUE;

		ELSE

			gSuperTrak.skill.Outfeed.state.stateMachine.stateTransition.start := FALSE;

		END_IF;

		IF gSuperTrak.skill.Outfeed.state.stateMachine.operationalState = COMPLETE THEN

			gSuperTrak.skill.Outfeed.state.stateMachine.stateTransition.reset := TRUE;
			StTargetExt_[7].ReleaseToTarget := TRUE;

		END_IF;

	END_IF;

	IF EDGENEG(StTargetExt_[7].PalletPresent) THEN

		StTargetExt_[7].ReleaseToTarget := FALSE;

	END_IF;

	//Virtual Target
	IF StTargetExt_[8].PalletPresent THEN

		StTargetExt_[8].ReleaseToTarget := TRUE;

	END_IF;

	IF EDGENEG(StTargetExt_[8].PalletPresent) THEN

		StTargetExt_[8].ReleaseToTarget := FALSE;

	END_IF;

	TON_Check_Parking ();

END_ACTION
```

#### ST_Events_Data.st
```iecst
ACTION ST_Events_Data:
	(*Define Event_Messages here*)

	(*Errors/Events are defined through a structure containing 5 different datas*)

	(* Severity, facility in which the event is being detected, code of the error, Event_Message for it and the ID generated for the Event*)
	Events[0].Severity_Code 	:= arEVENTLOG_SEVERITY_INFO;
	Events[0].Facility_Code 	:= 0;
	Events[0].Code_Value		:= 0;
	Events[0].Event_Message		:= 'SuperTrak Initialized Correctly';

	Events[1].Severity_Code 	:= arEVENTLOG_SEVERITY_ERROR;
	Events[1].Facility_Code 	:= 0;
	Events[1].Code_Value		:= 1;
	Events[1].Event_Message		:= 'Critical Hardware Error - Sections were not enabled';

	Events[2].Severity_Code 	:= arEVENTLOG_SEVERITY_ERROR;
	Events[2].Facility_Code 	:= 0;
	Events[2].Code_Value		:= 2;
	Events[2].Event_Message		:= 'Critical Hardware Error - Shuttles not recognized.';

	Events[3].Severity_Code 	:= arEVENTLOG_SEVERITY_ERROR;
	Events[3].Facility_Code 	:= 0;
	Events[3].Code_Value		:= 3;
	Events[3].Event_Message		:= 'Critical Hardware Error - Targets not enabled.';

	Events[4].Severity_Code 	:= arEVENTLOG_SEVERITY_ERROR;
	Events[4].Facility_Code 	:= 15;
	Events[4].Code_Value		:= 4;
	Events[4].Event_Message		:= 'Timeout Error - Lost connection to MES.';

(*	Change angel
	Events[5].Severity_Code 	:= arEVENTLOG_SEVERITY_ERROR;
	Events[5].Facility_Code 	:= 15;
	Events[5].Code_Value		:= 5;
	Events[5].Event_Message		:= 'Critical Error - Emergency Stop.';
*)
	Events[6].Severity_Code 	:= arEVENTLOG_SEVERITY_WARNING;
	Events[6].Facility_Code 	:= 0;
	Events[6].Code_Value		:= 6;
	Events[6].Event_Message		:= 'Timeout Error - Lost connection to Process Simulator.';

	Events[7].Severity_Code 	:= arEVENTLOG_SEVERITY_ERROR;
	Events[7].Facility_Code 	:= 0;
	Events[7].Code_Value		:= 7;
	Events[7].Event_Message		:= 'Timeout Error - Clearing Process Timed Out, Aborting process';

	Events[8].Severity_Code 	:= arEVENTLOG_SEVERITY_ERROR;
	Events[8].Facility_Code 	:= 0;
	Events[8].Code_Value		:= 8;
	Events[8].Event_Message		:= 'Number of SECTIONS is greater than maximum allowed';

	Events[9].Severity_Code 	:= arEVENTLOG_SEVERITY_ERROR;
	Events[9].Facility_Code 	:= 0;
	Events[9].Code_Value		:= 9;
	Events[9].Event_Message		:= 'Number of SHUTTLES is greater than maximum allowed';

	Events[10].Severity_Code 	:= arEVENTLOG_SEVERITY_ERROR;
	Events[10].Facility_Code 	:= 0;
	Events[10].Code_Value		:= 10;
	Events[10].Event_Message	:= 'Number of TARGETS is greater than maximum allowed';

	(* =========================================================================== *)
	(* SuperTrak Info *)

	Events[11].Severity_Code 	:= arEVENTLOG_SEVERITY_INFO;
	Events[11].Facility_Code 	:= 0;
	Events[11].Code_Value		:= 11;
	Events[11].Event_Message	:= 'SuperTrak State - Idle.';

	Events[12].Severity_Code 	:= arEVENTLOG_SEVERITY_INFO;
	Events[12].Facility_Code 	:= 0;
	Events[12].Code_Value		:= 12;
	Events[12].Event_Message	:= 'SuperTrak State - Starting.';

	Events[13].Severity_Code 	:= arEVENTLOG_SEVERITY_INFO;
	Events[13].Facility_Code 	:= 0;
	Events[13].Code_Value		:= 13;
	Events[13].Event_Message	:= 'SuperTrak State - Running.';

	Events[14].Severity_Code 	:= arEVENTLOG_SEVERITY_INFO;
	Events[14].Facility_Code 	:= 0;
	Events[14].Code_Value		:= 14;
	Events[14].Event_Message	:= 'SuperTrak State - Pausing.';

	Events[15].Severity_Code 	:= arEVENTLOG_SEVERITY_INFO;
	Events[15].Facility_Code 	:= 0;
	Events[15].Code_Value		:= 15;
	Events[15].Event_Message	:= 'SuperTrak State - Paused.';

	Events[16].Severity_Code 	:= arEVENTLOG_SEVERITY_INFO;
	Events[16].Facility_Code 	:= 0;
	Events[16].Code_Value		:= 16;
	Events[16].Event_Message	:= 'SuperTrak State - Suspending.';

	Events[17].Severity_Code 	:= arEVENTLOG_SEVERITY_INFO;
	Events[17].Facility_Code 	:= 0;
	Events[17].Code_Value		:= 17;
	Events[17].Event_Message	:= 'SuperTrak State - Suspended.';

	Events[18].Severity_Code 	:= arEVENTLOG_SEVERITY_INFO;
	Events[18].Facility_Code 	:= 0;
	Events[18].Code_Value		:= 18;
	Events[18].Event_Message	:= 'SuperTrak State - Unsuspending.';

	Events[19].Severity_Code 	:= arEVENTLOG_SEVERITY_INFO;
	Events[19].Facility_Code 	:= 0;
	Events[19].Code_Value		:= 19;
	Events[19].Event_Message	:= 'SuperTrak State - Holding.';

	Events[20].Severity_Code 	:= arEVENTLOG_SEVERITY_INFO;
	Events[20].Facility_Code 	:= 0;
	Events[20].Code_Value		:= 20;
	Events[20].Event_Message	:= 'SuperTrak State - Held.';

	Events[21].Severity_Code 	:= arEVENTLOG_SEVERITY_INFO;
	Events[21].Facility_Code 	:= 0;
	Events[21].Code_Value		:= 21;
	Events[21].Event_Message	:= 'SuperTrak State - Unholding.';

	Events[22].Severity_Code 	:= arEVENTLOG_SEVERITY_INFO;
	Events[22].Facility_Code 	:= 0;
	Events[22].Code_Value		:= 22;
	Events[22].Event_Message	:= 'SuperTrak State - Completing.';

	Events[23].Severity_Code 	:= arEVENTLOG_SEVERITY_INFO;
	Events[23].Facility_Code 	:= 0;
	Events[23].Code_Value		:= 23;
	Events[23].Event_Message	:= 'SuperTrak State - Complete.';

	Events[24].Severity_Code 	:= arEVENTLOG_SEVERITY_INFO;
	Events[24].Facility_Code 	:= 0;
	Events[24].Code_Value		:= 24;
	Events[24].Event_Message	:= 'SuperTrak State - Resetting.';

	Events[25].Severity_Code 	:= arEVENTLOG_SEVERITY_INFO;
	Events[25].Facility_Code 	:= 0;
	Events[25].Code_Value		:= 25;
	Events[25].Event_Message	:= 'SuperTrak State - Stopping.';

	Events[26].Severity_Code 	:= arEVENTLOG_SEVERITY_INFO;
	Events[26].Facility_Code 	:= 0;
	Events[26].Code_Value		:= 26;
	Events[26].Event_Message	:= 'SuperTrak State - Stopped.';

	Events[27].Severity_Code 	:= arEVENTLOG_SEVERITY_INFO;
	Events[27].Facility_Code 	:= 0;
	Events[27].Code_Value		:= 27;
	Events[27].Event_Message	:= 'SuperTrak State - Aborting.';

	Events[28].Severity_Code 	:= arEVENTLOG_SEVERITY_INFO;
	Events[28].Facility_Code 	:= 0;
	Events[28].Code_Value		:= 28;
	Events[28].Event_Message	:= 'SuperTrak State - Aborted.';

	Events[29].Severity_Code 	:= arEVENTLOG_SEVERITY_INFO;
	Events[29].Facility_Code 	:= 0;
	Events[29].Code_Value		:= 29;
	Events[29].Event_Message	:= 'SuperTrak State - Clearing.';

	(************************************************************************************)
	(*Shuttles Critical Events*)

	FOR i := 1 TO SUPERTRAK_SHUTTLES DO
		iEvent := i+29;

		Events[iEvent].Severity_Code 	:= arEVENTLOG_SEVERITY_ERROR;
		Events[iEvent].Facility_Code 	:= 0;
		Events[iEvent].Code_Value		:= iEvent;
		Events[iEvent].Event_Message	:='Skill moveShuttle.- Final Target does not exist';

	END_FOR;

	FOR i := 1 TO SUPERTRAK_SHUTTLES DO
		iEvent := i+41;

		Events[iEvent].Severity_Code 	:= arEVENTLOG_SEVERITY_INFO;
		Events[iEvent].Facility_Code 	:= 0;
		Events[iEvent].Code_Value		:= iEvent;
		Events[iEvent].Event_Message	:= 'Skill moveShuttle.-  Shuttle finished product cycle.';

	END_FOR;

	FOR i := 1 TO SUPERTRAK_SHUTTLES DO
		iEvent := i+53;

		Events[iEvent].Severity_Code 	:= arEVENTLOG_SEVERITY_ERROR;
		Events[iEvent].Facility_Code 	:= 0;
		Events[iEvent].Code_Value		:= iEvent;
		Events[iEvent].Event_Message	:= 'Skill moveShuttle.-  Final Target equals current target.';

	END_FOR;

	FOR i := 1 TO SUPERTRAK_SHUTTLES DO
		iEvent := i+65;

		Events[iEvent].Severity_Code 	:= arEVENTLOG_SEVERITY_ERROR;
		Events[iEvent].Facility_Code 	:= 0;
		Events[iEvent].Code_Value		:= iEvent;
		Events[iEvent].Event_Message	:= 'Skill moveShuttle.-  Skill was aborted.';

	END_FOR;

	Events[77].Severity_Code 	:= arEVENTLOG_SEVERITY_ERROR;
	Events[77].Facility_Code 	:= 15;
	Events[77].Code_Value		:= 77;
	Events[77].Event_Message	:= 'Skill checkParking.- Skill was aborted';

	(*Service Stations Events*)

	Events[78].Severity_Code 	:= arEVENTLOG_SEVERITY_ERROR;
	Events[78].Facility_Code 	:= 15;
	Events[78].Code_Value		:= 78;
	Events[78].Event_Message	:= 'Light Barrier detected illegal access. System Aborted.';

	Events[79].Severity_Code 	:= arEVENTLOG_SEVERITY_ERROR;
	Events[79].Facility_Code 	:= 15;
	Events[79].Code_Value		:= 79;
	Events[79].Event_Message	:= 'QA Service door was illegaly opened';

	Events[80].Severity_Code 	:= arEVENTLOG_SEVERITY_WARNING;
	Events[80].Facility_Code 	:= 0;
	Events[80].Code_Value		:= 80;
	Events[80].Event_Message	:= 'Outfeed storage is full, please take the products out to continue';

	Events[81].Severity_Code 	:= arEVENTLOG_SEVERITY_SUCCESS;
	Events[81].Facility_Code 	:= 0;
	Events[81].Code_Value		:= 81;
	Events[81].Event_Message	:= 'Maintenance Mode - Outfeed clearing, restoring the process';

	Events[82].Severity_Code 	:= arEVENTLOG_SEVERITY_WARNING;
	Events[82].Facility_Code 	:= 0;
	Events[82].Code_Value		:= 82;
	Events[82].Event_Message	:= 'SuperTrak process stopped';

	Events[83].Severity_Code 	:= arEVENTLOG_SEVERITY_WARNING;
	Events[83].Facility_Code 	:= 0;
	Events[83].Code_Value		:= 83;
	Events[83].Event_Message	:= 'Error has not yet been acknowledged, clear transition not possible';

	Events[84].Severity_Code 	:= arEVENTLOG_SEVERITY_SUCCESS;
	Events[84].Facility_Code 	:= 0;
	Events[84].Code_Value		:= 84;
	Events[84].Event_Message	:= 'Refill succesfully finished';

	(* Definition of all events ID's *)
	FOR i := 0 TO 99 DO
		Events[i].ID := ArEventLogMakeEventID(Severity := Events[i].Severity_Code , Facility := Events[i].Facility_Code , ErrorCode := Events[i].Code_Value);
	END_FOR;

END_ACTION
```

#### Assem_Events_Data.st
```iecst
ACTION Assembly_Events_Data:

	(*Errors/Events are defined through a structure containing 5 different datas*)

	(* Severity, facility in which the event is being detected, code of the error, Event_Message for it and the ID generated for the Event*)

	(***************************************************************************************)

	Events[100].Severity_Code 	:= arEVENTLOG_SEVERITY_ERROR;
	Events[100].Facility_Code 	:= 0;
	Events[100].Code_Value		:= 100;
	Events[100].Event_Message	:= 'Timeout Error - Clearing failed.';

	Events[101].Severity_Code 	:= arEVENTLOG_SEVERITY_ERROR;
	Events[101].Facility_Code 	:= 0;
	Events[101].Code_Value		:= 101;
	Events[101].Event_Message	:= 'Comau Illegal Position.';

	Events[102].Severity_Code 	:= arEVENTLOG_SEVERITY_ERROR;
	Events[102].Facility_Code 	:= 15;
	Events[102].Code_Value		:= 102;
	Events[102].Event_Message	:= 'Critical Hardware Error - Paper Cups Supply not supported';

	Events[103].Severity_Code 	:= arEVENTLOG_SEVERITY_ERROR;
	Events[103].Facility_Code 	:= 0;
	Events[103].Code_Value		:= 103;
	Events[103].Event_Message	:= 'Critical Hardware Error -';

	Events[104].Severity_Code 	:= arEVENTLOG_SEVERITY_ERROR;
	Events[104].Facility_Code 	:= 15;
	Events[104].Code_Value		:= 104;
	Events[104].Event_Message	:= 'Timeout Error - Lost connection to MES.';

	Events[105].Severity_Code 	:= arEVENTLOG_SEVERITY_ERROR;
	Events[105].Facility_Code 	:= 15;
	Events[105].Code_Value		:= 105;
	Events[105].Event_Message	:= 'Critical Error - Emergency Stop.';

	Events[106].Severity_Code 	:= arEVENTLOG_SEVERITY_WARNING;
	Events[106].Facility_Code 	:= 0;
	Events[106].Code_Value		:= 106;
	Events[106].Event_Message	:= 'Timeout Error - Lost connection to Process Simulator.';

	(***************************************************************************************)

	(*Skills Events*)

	Events[107].Severity_Code 	:= arEVENTLOG_SEVERITY_ERROR;
	Events[107].Facility_Code 	:= 0;
	Events[107].Code_Value		:= 107;
	Events[107].Event_Message	:= 'goHome Skill was aborted';

	Events[108].Severity_Code 	:= arEVENTLOG_SEVERITY_ERROR;
	Events[108].Facility_Code 	:= 0;
	Events[108].Code_Value		:= 108;
	Events[108].Event_Message	:= 'provideCup Skill was aborted';

	Events[109].Severity_Code 	:= arEVENTLOG_SEVERITY_ERROR;
	Events[109].Facility_Code 	:= 0;
	Events[109].Code_Value		:= 109;
	Events[109].Event_Message	:= 'providePellet Skill was aborted';

	(***************************************************************************************)
	(* Assembly Info states*)

	Events[111].Severity_Code 	:= arEVENTLOG_SEVERITY_INFO;
	Events[111].Facility_Code 	:= 0;
	Events[111].Code_Value		:= 111;
	Events[111].Event_Message	:= 'Assembly State - Idle.';

	Events[112].Severity_Code 	:= arEVENTLOG_SEVERITY_INFO;
	Events[112].Facility_Code 	:= 0;
	Events[112].Code_Value		:= 112;
	Events[112].Event_Message	:= 'Assembly State - Starting.';

	Events[113].Severity_Code 	:= arEVENTLOG_SEVERITY_INFO;
	Events[113].Facility_Code 	:= 0;
	Events[113].Code_Value		:= 113;
	Events[113].Event_Message	:= 'Assembly State - Running.';

	Events[114].Severity_Code 	:= arEVENTLOG_SEVERITY_INFO;
	Events[114].Facility_Code 	:= 0;
	Events[114].Code_Value		:= 114;
	Events[114].Event_Message	:= 'Assembly State - Pausing.';

	Events[115].Severity_Code 	:= arEVENTLOG_SEVERITY_INFO;
	Events[115].Facility_Code 	:= 0;
	Events[115].Code_Value		:= 115;
	Events[115].Event_Message	:= 'Assembly State - Paused.';

	Events[116].Severity_Code 	:= arEVENTLOG_SEVERITY_INFO;
	Events[116].Facility_Code 	:= 0;
	Events[116].Code_Value		:= 116;
	Events[116].Event_Message	:= 'Assembly State - Suspending.';

	Events[117].Severity_Code 	:= arEVENTLOG_SEVERITY_INFO;
	Events[117].Facility_Code 	:= 0;
	Events[117].Code_Value		:= 117;
	Events[117].Event_Message	:= 'Assembly State - Suspended.';

	Events[118].Severity_Code 	:= arEVENTLOG_SEVERITY_INFO;
	Events[118].Facility_Code 	:= 0;
	Events[118].Code_Value		:= 118;
	Events[118].Event_Message	:= 'Assembly State - Unsuspending.';

	Events[119].Severity_Code 	:= arEVENTLOG_SEVERITY_INFO;
	Events[119].Facility_Code 	:= 0;
	Events[119].Code_Value		:= 119;
	Events[119].Event_Message	:= 'Assembly State - Holding.';

	Events[120].Severity_Code 	:= arEVENTLOG_SEVERITY_INFO;
	Events[120].Facility_Code 	:= 0;
	Events[120].Code_Value		:= 120;
	Events[120].Event_Message	:= 'Assembly State - Held.';

	Events[121].Severity_Code 	:= arEVENTLOG_SEVERITY_INFO;
	Events[121].Facility_Code 	:= 0;
	Events[121].Code_Value		:= 121;
	Events[121].Event_Message	:= 'Assembly State - Unholding.';

	Events[122].Severity_Code 	:= arEVENTLOG_SEVERITY_INFO;
	Events[122].Facility_Code 	:= 0;
	Events[122].Code_Value		:= 122;
	Events[122].Event_Message	:= 'Assembly State - Completing.';

	Events[123].Severity_Code 	:= arEVENTLOG_SEVERITY_INFO;
	Events[123].Facility_Code 	:= 0;
	Events[123].Code_Value		:= 123;
	Events[123].Event_Message	:= 'Assembly State - Complete.';

	Events[124].Severity_Code 	:= arEVENTLOG_SEVERITY_INFO;
	Events[124].Facility_Code 	:= 0;
	Events[124].Code_Value		:= 124;
	Events[124].Event_Message	:= 'Assembly State - Resetting.';

	Events[125].Severity_Code 	:= arEVENTLOG_SEVERITY_INFO;
	Events[125].Facility_Code 	:= 0;
	Events[125].Code_Value		:= 125;
	Events[125].Event_Message	:= 'Assembly State - Stopping.';

	Events[126].Severity_Code 	:= arEVENTLOG_SEVERITY_INFO;
	Events[126].Facility_Code 	:= 0;
	Events[126].Code_Value		:= 126;
	Events[126].Event_Message	:= 'Assembly State - Stopped.';

	Events[127].Severity_Code 	:= arEVENTLOG_SEVERITY_INFO;
	Events[127].Facility_Code 	:= 0;
	Events[127].Code_Value		:= 127;
	Events[127].Event_Message	:= 'Assembly State - Aborting.';

	Events[128].Severity_Code 	:= arEVENTLOG_SEVERITY_INFO;
	Events[128].Facility_Code 	:= 0;
	Events[128].Code_Value		:= 128;
	Events[128].Event_Message	:= 'Assembly State - Aborted.';

	Events[129].Severity_Code 	:= arEVENTLOG_SEVERITY_INFO;
	Events[129].Facility_Code 	:= 0;
	Events[129].Code_Value		:= 129;
	Events[129].Event_Message	:= 'Assembly State - Clearing.';

	(***************************************************************************************)

	(*Service Stations Events*)

	Events[130].Severity_Code 	:= arEVENTLOG_SEVERITY_WARNING;
	Events[130].Facility_Code 	:= 15;
	Events[130].Code_Value		:= 130;
	Events[130].Event_Message	:= 'Maintenance Mode - Requested by the user';

	Events[131].Severity_Code 	:= arEVENTLOG_SEVERITY_ERROR;
	Events[131].Facility_Code 	:= 0;
	Events[131].Code_Value		:= 131;
	Events[131].Event_Message	:= 'Error in the Homing Procedure';

	Events[132].Severity_Code 	:= arEVENTLOG_SEVERITY_WARNING;
	Events[132].Facility_Code 	:= 15;
	Events[132].Code_Value		:= 132;
	Events[132].Event_Message	:= 'Maintenance Mode - Plastic Cup ordered, but there were any in the tray';

	Events[133].Severity_Code 	:= arEVENTLOG_SEVERITY_SUCCESS;
	Events[133].Facility_Code 	:= 15;
	Events[133].Code_Value		:= 133;
	Events[133].Event_Message	:= 'Maintenance Mode - Refill finished, restoring the process';
	(***************************************************************************************)

	(*door sensors and magnets Events*)

	Events[140].Severity_Code 	:= arEVENTLOG_SEVERITY_ERROR;
	Events[140].Facility_Code 	:= 15;
	Events[140].Code_Value		:= 140;
	Events[140].Event_Message	:= 'Assembly Door was illegally opened';

	Events[141].Severity_Code 	:= arEVENTLOG_SEVERITY_SUCCESS;
	Events[141].Facility_Code 	:= 15;
	Events[141].Code_Value		:= 141;
	Events[141].Event_Message	:= 'Refill succesfully finished';

	Events[142].Severity_Code 	:= arEVENTLOG_SEVERITY_ERROR;
	Events[142].Facility_Code 	:= 15;
	Events[142].Code_Value		:= 142;
	Events[142].Event_Message	:= 'Assembly Paper Tray Right Door was illegally opened';

	Events[143].Severity_Code 	:= arEVENTLOG_SEVERITY_ERROR;
	Events[143].Facility_Code 	:= 15;
	Events[143].Code_Value		:= 143;
	Events[143].Event_Message	:= 'Assembly Paper Tray Left Door was illegally opened';

	Events[144].Severity_Code 	:= arEVENTLOG_SEVERITY_ERROR;
	Events[144].Facility_Code 	:= 15;
	Events[144].Code_Value		:= 144;
	Events[144].Event_Message	:= 'Assembly Plastic Tray drawer was illegally opened';

	Events[145].Severity_Code 	:= arEVENTLOG_SEVERITY_ERROR;
	Events[145].Facility_Code 	:= 15;
	Events[145].Code_Value		:= 145;
	Events[145].Event_Message	:= 'Assembly Paper Tray drawer was illegally opened';

(***************************************************************************************)

	Events[182].Severity_Code 	:= arEVENTLOG_SEVERITY_WARNING;
	Events[182].Facility_Code 	:= 0;
	Events[182].Code_Value		:= 182;
	Events[182].Event_Message	:= 'Assembly process stopped';

	Events[183].Severity_Code 	:= arEVENTLOG_SEVERITY_ERROR;
	Events[183].Facility_Code 	:= 0;
	Events[183].Code_Value		:= 183;
	Events[183].Event_Message	:= '';

	(* Definition of all events ID's *)
	FOR i := 100 TO 199 DO
		Events[i].ID := ArEventLogMakeEventID(Severity := Events[i].Severity_Code , Facility := Events[i].Facility_Code , ErrorCode := Events[i].Code_Value);
	END_FOR;

END_ACTION
```

### Program Logical/Events_handling/EventLoggerMNG

#### Main.st
```iecst
 (*******************************************************************
 * Implementation of program EventLog
 ********************************************************************)

PROGRAM _INIT
	strcpy(ADR(EventLog.Event.AdditionalData),ADR('This is an information entry from the user, which could contain anything up to the length being written in this message.'));
	EventLog.Event.AdditionalDataSize := strlen(ADR(EventLog.Event.AdditionalData)) + 1;
	EventLog.Event.AdditionalDataFormat := arEVENTLOG_ADDFORMAT_TEXT;
	(*See ArEventLog help for the description of the event id, facilities 0-15 are reserved for customer use.*)

	(* We first try to delete the logger, then create it again, and if the creation works correctly we will receive a successs message through the logger *)
	ST_Last_Info_Written := 0;
	Assembly_Last_Info_Written := 0;
	General_Last_Info_Written := 0;
	EventLog.Commands.CreateUserLog := TRUE;
	Event_Code := 250;
	EventLog.Commands.WriteUserEvent := TRUE;
END_PROGRAM

PROGRAM _CYCLIC

	CASE EventLog.Data.Step OF
		(*Waits for user input (command).*)
		STEP_WAIT_FOR_INPUT:

			IF EventLog.Commands.DeleteUserLog THEN
				EventLog.Commands.DeleteUserLog := FALSE;
				EventLog.Data.Step := STEP_GET_LOGBOOK_IDENT;
				EventLog.Data.GetIdentFailNextStep := STEP_ERROR;
				EventLog.Data.GetIdentOkNextStep := STEP_DELETE_LOGBOOK;
			ELSIF EventLog.Commands.CreateUserLog THEN
				EventLog.Commands.CreateUserLog := FALSE;
				EventLog.Data.Step := STEP_GET_LOGBOOK_IDENT;
				EventLog.Data.GetIdentFailNextStep := STEP_CREATE_LOGBOOK;
				EventLog.Data.GetIdentOkNextStep := STEP_WAIT_FOR_INPUT;
			ELSIF EventLog.Commands.ReadLatestEvent THEN
				EventLog.Commands.ReadLatestEvent := FALSE;
				EventLog.Data.Step := STEP_GET_LOGBOOK_IDENT;
				EventLog.Data.GetIdentFailNextStep := STEP_ERROR;
				EventLog.Data.GetIdentOkNextStep := STEP_GET_LATEST_RECORD_ID;
			ELSIF EventLog.Commands.WriteUserEvent THEN

				(*Definition of the message before writting it to be sure a knew event_ID will not overwrite it*)
				EventLog.FunctionBlocks.ArEventLogWrite_0.EventID := Events[Event_Code].ID;
				EventLog.FunctionBlocks.ArEventLogWrite_0.AddData := ADR(Events[Event_Code].Event_Message);

				(*Detection of info messages*)
				IF Events[Event_Code].Severity_Code = arEVENTLOG_SEVERITY_INFO THEN
					Info_Event := TRUE;
				ELSE
					Info_Event := FALSE;
				END_IF;

				(*We only write in the logger if the message we are about to write is not the last one written or if the las info message written in the logger is not the one we are trying to write now*)
				IF (Event_Code <> Last_Event_Written AND NOT Info_Event) OR
					(Info_Event AND (Event_Code <> ST_Last_Info_Written AND Event_Code <> Assembly_Last_Info_Written AND General_Last_Info_Written <> Event_Code))
					THEN
					EventLog.Commands.WriteUserEvent := FALSE;
					EventLog.Data.Step := STEP_GET_LOGBOOK_IDENT;
					EventLog.Data.GetIdentFailNextStep := STEP_ERROR;
					EventLog.Data.GetIdentOkNextStep := STEP_WRITE_EVENT;
				ELSE
					EventLog.Commands.WriteUserEvent := FALSE;
					EventLog.Data.Step := STEP_WAIT_FOR_INPUT;
				END_IF;

			ELSIF EventLog.Commands.ReadPreviousEvent THEN
				EventLog.Commands.ReadPreviousEvent := FALSE;
				EventLog.Data.Step := STEP_GET_LOGBOOK_IDENT;
				EventLog.Data.GetIdentFailNextStep := STEP_ERROR;
				EventLog.Data.GetIdentOkNextStep := STEP_GET_PREVIOUS_RECORD_ID;
			END_IF

			(*Gets the ident of the user logbook "STEvents".*)
		STEP_GET_LOGBOOK_IDENT:

			IF EventLog.FunctionBlocks.ArEventLogGetIdent_0.Done THEN
				EventLog.FunctionBlocks.ArEventLogGetIdent_0.Execute := FALSE;
				EventLog.Data.Ident := EventLog.FunctionBlocks.ArEventLogGetIdent_0.Ident;
				EventLog.Data.StatusID := ERR_OK;
				EventLog.Data.Step := EventLog.Data.GetIdentOkNextStep;
			ELSIF EventLog.FunctionBlocks.ArEventLogGetIdent_0.Error THEN
				EventLog.FunctionBlocks.ArEventLogGetIdent_0.Execute := FALSE;
				EventLog.Data.StatusID := EventLog.FunctionBlocks.ArEventLogGetIdent_0.StatusID;
				EventLog.Data.Step := EventLog.Data.GetIdentFailNextStep;
			ELSE
				(*Execute the FB only if the ident isn't already set.*)
				IF EventLog.Data.Ident = 0 THEN
					EventLog.FunctionBlocks.ArEventLogGetIdent_0.Name := 'UsrEvLog';
					EventLog.FunctionBlocks.ArEventLogGetIdent_0.Execute := TRUE;
				ELSE
					EventLog.Data.StatusID := ERR_OK;
					EventLog.Data.Step := EventLog.Data.GetIdentOkNextStep;
				END_IF
			END_IF

			(*Creates the user logbook "UsrEvLog".*)
		STEP_CREATE_LOGBOOK:
			IF EventLog.FunctionBlocks.ArEventLogCreate_0.Done THEN
				EventLog.FunctionBlocks.ArEventLogCreate_0.Execute := FALSE;
				EventLog.Data.Ident := EventLog.FunctionBlocks.ArEventLogCreate_0.Ident;
				EventLog.Data.StatusID := ERR_OK;
				EventLog.Data.Step := STEP_WAIT_FOR_INPUT;
			ELSIF EventLog.FunctionBlocks.ArEventLogCreate_0.Error THEN
				EventLog.FunctionBlocks.ArEventLogCreate_0.Execute := FALSE;
				EventLog.Data.StatusID := EventLog.FunctionBlocks.ArEventLogCreate_0.StatusID;
				EventLog.Data.Step := STEP_ERROR;
			ELSE
				EventLog.FunctionBlocks.ArEventLogCreate_0.Name := 'UsrEvLog';
				EventLog.FunctionBlocks.ArEventLogCreate_0.Size := 10000;
				EventLog.FunctionBlocks.ArEventLogCreate_0.Persistence := arEVENTLOG_PERSISTENCE_VOLATILE;
				EventLog.FunctionBlocks.ArEventLogCreate_0.Info := 0;
				EventLog.FunctionBlocks.ArEventLogCreate_0.Execute := TRUE;
			END_IF

			(*Deletes the user logbook "UsrEvLog".*)
		STEP_DELETE_LOGBOOK:
			IF EventLog.FunctionBlocks.ArEventLogDelete_0.Done THEN
				EventLog.FunctionBlocks.ArEventLogDelete_0.Execute := FALSE;
				EventLog.Data.Ident := 0;
				EventLog.Data.StatusID := ERR_OK;
				EventLog.Data.Step := STEP_WAIT_FOR_INPUT;
			ELSIF EventLog.FunctionBlocks.ArEventLogDelete_0.Error THEN
				EventLog.FunctionBlocks.ArEventLogDelete_0.Execute := FALSE;
				EventLog.Data.StatusID := EventLog.FunctionBlocks.ArEventLogDelete_0.StatusID;
				EventLog.Data.Step := STEP_ERROR;
			ELSE
				EventLog.FunctionBlocks.ArEventLogDelete_0.Ident := EventLog.Data.Ident;
				EventLog.FunctionBlocks.ArEventLogDelete_0.Execute := TRUE;
			END_IF

			(*Writes the event set in EventLog.Event to the user logbook "UsrEvLog".*)
		STEP_WRITE_EVENT:
			IF EventLog.FunctionBlocks.ArEventLogWrite_0.Done THEN
				EventLog.FunctionBlocks.ArEventLogWrite_0.Execute := FALSE;
				EventLog.Data.StatusID := ERR_OK;

				New_Event := TRUE;
				EventLog.Data.Step := STEP_WAIT_FOR_INPUT;
			ELSIF EventLog.FunctionBlocks.ArEventLogWrite_0.Error THEN
				EventLog.FunctionBlocks.ArEventLogWrite_0.Execute := FALSE;
				EventLog.Data.StatusID := EventLog.FunctionBlocks.ArEventLogWrite_0.StatusID;
				EventLog.Data.Step := STEP_ERROR;
			ELSE

				(* Identification of the module generating the new entry *)
				IF Event_Code < 100 THEN
					EventLog.Event.EnteredBy := 'SuperTrak';
				ELSIF Event_Code < 200 THEN
					EventLog.Event.EnteredBy := 'Assembly';
				ELSE
					EventLog.Event.EnteredBy := 'General Msg';
				END_IF;

				(* Then the defintion for the rest of the message parameters is made *)
				EventLog.FunctionBlocks.ArEventLogWrite_0.Ident := EventLog.Data.Ident;
				EventLog.Event.Customer							  := TRUE;
				EventLog.FunctionBlocks.ArEventLogWrite_0.TimeStamp := 0; (*System timestamp.*)
				EventLog.FunctionBlocks.ArEventLogWrite_0.ObjectID := EventLog.Event.EnteredBy;
				EventLog.FunctionBlocks.ArEventLogWrite_0.OriginRecordID := EventLog.Event.OriginID;
				EventLog.FunctionBlocks.ArEventLogWrite_0.AddDataFormat := EventLog.Event.AdditionalDataFormat;
				EventLog.FunctionBlocks.ArEventLogWrite_0.AddDataSize := EventLog.Event.AdditionalDataSize;
				(* The writing is executed *)
				EventLog.FunctionBlocks.ArEventLogWrite_0.Execute := TRUE;

			END_IF;

			(*Gets the id of the latest record in the user logbook "UsrEvLog".*)
		STEP_GET_LATEST_RECORD_ID:
			IF EventLog.FunctionBlocks.ArEventLogGetLatestRecordID_0.Done THEN
				EventLog.FunctionBlocks.ArEventLogGetLatestRecordID_0.Execute := FALSE;
				EventLog.Event.RecordID := EventLog.FunctionBlocks.ArEventLogGetLatestRecordID_0.RecordID;
				EventLog.Data.StatusID := ERR_OK;
				EventLog.Data.Step := STEP_READ_EVENT;
			ELSIF EventLog.FunctionBlocks.ArEventLogGetLatestRecordID_0.Error THEN
				EventLog.FunctionBlocks.ArEventLogGetLatestRecordID_0.Execute := FALSE;
				EventLog.Data.StatusID := EventLog.FunctionBlocks.ArEventLogGetLatestRecordID_0.StatusID;
				EventLog.Data.Step := STEP_ERROR;
			ELSE
				EventLog.FunctionBlocks.ArEventLogGetLatestRecordID_0.Ident := EventLog.Data.Ident;
				EventLog.FunctionBlocks.ArEventLogGetLatestRecordID_0.Execute := TRUE;
			END_IF

			(*Gets the id of the previous record of the given record id (EventLog.Event.RecordID).*)
		STEP_GET_PREVIOUS_RECORD_ID:
			IF EventLog.FunctionBlocks.ArEventLogGetPreviousRecordID_0.Done THEN
				EventLog.FunctionBlocks.ArEventLogGetPreviousRecordID_0.Execute := FALSE;
				EventLog.Event.RecordID := EventLog.FunctionBlocks.ArEventLogGetPreviousRecordID_0.PrevRecordID;
				EventLog.Data.StatusID := ERR_OK;
				EventLog.Data.Step := STEP_READ_EVENT;
			ELSIF EventLog.FunctionBlocks.ArEventLogGetPreviousRecordID_0.Error THEN
				EventLog.FunctionBlocks.ArEventLogGetPreviousRecordID_0.Execute := FALSE;
				EventLog.Data.StatusID := EventLog.FunctionBlocks.ArEventLogGetPreviousRecordID_0.StatusID;
				EventLog.Data.Step := STEP_ERROR;
			ELSE
				EventLog.FunctionBlocks.ArEventLogGetPreviousRecordID_0.Ident := EventLog.Data.Ident;
				EventLog.FunctionBlocks.ArEventLogGetPreviousRecordID_0.RecordID := EventLog.Event.RecordID;
				EventLog.FunctionBlocks.ArEventLogGetPreviousRecordID_0.Execute := TRUE;
			END_IF

			(*Reads the event with the given record id from the to user logbook "UsrEvLog".*)
		STEP_READ_EVENT:
			IF EventLog.FunctionBlocks.ArEventLogRead_0.Done THEN
				EventLog.FunctionBlocks.ArEventLogRead_0.Execute := FALSE;
				EventLog.Event.AdditionalDataFormat := EventLog.FunctionBlocks.ArEventLogRead_0.AddDataFormat;
				EventLog.Event.AdditionalDataSize := EventLog.FunctionBlocks.ArEventLogRead_0.AddDataSize;
				EventLog.Event.TimeStamp := EventLog.FunctionBlocks.ArEventLogRead_0.TimeStamp;
				EventLog.Event.OriginID := EventLog.FunctionBlocks.ArEventLogRead_0.OriginRecordID;
				EventLog.Data.StatusID := ERR_OK;
				EventLog.Event.ErrorNumber := 0;
				EventLog.Event.Customer := ArEventLogIsCustomerArea(EventID := EventLog.FunctionBlocks.ArEventLogRead_0.EventID);
				EventLog.Event.Severity := GetSeverity(EventID := EventLog.FunctionBlocks.ArEventLogRead_0.EventID);
				EventLog.Event.Code := GetCode(EventID := EventLog.FunctionBlocks.ArEventLogRead_0.EventID);
				EventLog.Event.Facility := GetFacility(EventID := EventLog.FunctionBlocks.ArEventLogRead_0.EventID);
				IF EventLog.FunctionBlocks.ArEventLogRead_0.StatusID = arEVENTLOG_WRN_NO_EVENTID THEN
					(*The given record id is not an event id record. Invoke ArEventLogReadErrorNumber to read the error number and the severity.*)
					EventLog.Data.Step := STEP_READ_ERROR_NUMBER;
				ELSIF EventLog.Event.AdditionalDataSize > 0 THEN
					EventLog.Data.Step := STEP_READ_ADDITIONAL_DATA;
				ELSE
					EventLog.Data.Step := STEP_READ_OBJECT_ID;
				END_IF
			ELSIF EventLog.FunctionBlocks.ArEventLogRead_0.Error THEN
				EventLog.FunctionBlocks.ArEventLogRead_0.Execute := FALSE;
				EventLog.Data.StatusID := EventLog.FunctionBlocks.ArEventLogRead_0.StatusID;
				EventLog.Data.Step := STEP_ERROR;
			ELSE
				EventLog.FunctionBlocks.ArEventLogRead_0.Ident := EventLog.Data.Ident;
				EventLog.FunctionBlocks.ArEventLogRead_0.RecordID := EventLog.Event.RecordID;
				EventLog.FunctionBlocks.ArEventLogRead_0.Execute := TRUE;
			END_IF

			(*Reads the error number event with the given record id from the user logbook "UsrEvLog".*)
		STEP_READ_ERROR_NUMBER:
			IF EventLog.FunctionBlocks.ArEventLogReadErrorNumber_0.Done THEN
				EventLog.FunctionBlocks.ArEventLogReadErrorNumber_0.Execute := FALSE;
				EventLog.Event.ErrorNumber := EventLog.FunctionBlocks.ArEventLogReadErrorNumber_0.ErrorNumber;
				EventLog.Event.Severity := EventLog.FunctionBlocks.ArEventLogReadErrorNumber_0.Severity;
				EventLog.Data.StatusID := ERR_OK;
				IF EventLog.Event.AdditionalDataSize > 0 THEN
					EventLog.Data.Step := STEP_READ_ADDITIONAL_DATA;
				ELSE
					EventLog.Data.Step := STEP_READ_OBJECT_ID;
				END_IF
			ELSIF EventLog.FunctionBlocks.ArEventLogReadErrorNumber_0.Error THEN
				EventLog.FunctionBlocks.ArEventLogReadErrorNumber_0.Execute := FALSE;
				EventLog.Data.StatusID := EventLog.FunctionBlocks.ArEventLogReadErrorNumber_0.StatusID;
				EventLog.Data.Step := STEP_ERROR;
			ELSE
				EventLog.FunctionBlocks.ArEventLogReadErrorNumber_0.Ident := EventLog.Data.Ident;
				EventLog.FunctionBlocks.ArEventLogReadErrorNumber_0.RecordID := EventLog.Event.RecordID;
				EventLog.FunctionBlocks.ArEventLogReadErrorNumber_0.Execute := TRUE;
			END_IF

			(*Reads the additional data of the event with the given record id from the user logbook "UsrEvLog".*)
		STEP_READ_ADDITIONAL_DATA:
			IF EventLog.FunctionBlocks.ArEventLogReadAddData_0.Done THEN
				EventLog.FunctionBlocks.ArEventLogReadAddData_0.Execute := FALSE;
				EventLog.Event.AdditionalDataSize := EventLog.FunctionBlocks.ArEventLogReadAddData_0.AddDataSize;
				EventLog.Data.StatusID := ERR_OK;
				EventLog.Data.Step := STEP_READ_OBJECT_ID;
			ELSIF EventLog.FunctionBlocks.ArEventLogReadAddData_0.Error THEN
				EventLog.FunctionBlocks.ArEventLogReadAddData_0.Execute := FALSE;
				EventLog.Data.StatusID := EventLog.FunctionBlocks.ArEventLogReadAddData_0.StatusID;
				EventLog.Data.Step := STEP_ERROR;
			ELSE
				EventLog.FunctionBlocks.ArEventLogReadAddData_0.Ident := EventLog.Data.Ident;
				EventLog.FunctionBlocks.ArEventLogReadAddData_0.RecordID := EventLog.Event.RecordID;
				EventLog.FunctionBlocks.ArEventLogReadAddData_0.BytesToRead := SIZEOF(EventLog.Event.AdditionalData);
				EventLog.FunctionBlocks.ArEventLogReadAddData_0.AddData := ADR(EventLog.Event.AdditionalData);
				EventLog.FunctionBlocks.ArEventLogReadAddData_0.Execute := TRUE;
			END_IF

			(*Reads the object id of the event with the given record id from the user logbook "UsrEvLog".*)
		STEP_READ_OBJECT_ID:
			IF EventLog.FunctionBlocks.ArEventLogReadObjectID_0.Done THEN
				EventLog.FunctionBlocks.ArEventLogReadObjectID_0.Execute := FALSE;
				EventLog.Event.EnteredBy := EventLog.FunctionBlocks.ArEventLogReadObjectID_0.ObjectID;
				EventLog.Data.StatusID := ERR_OK;
				EventLog.Data.Step := STEP_WAIT_FOR_INPUT;
			ELSIF EventLog.FunctionBlocks.ArEventLogReadObjectID_0.Error THEN
				EventLog.FunctionBlocks.ArEventLogReadObjectID_0.Execute := FALSE;
				EventLog.Data.StatusID := EventLog.FunctionBlocks.ArEventLogReadObjectID_0.StatusID;
				EventLog.Data.Step := STEP_ERROR;
			ELSE
				EventLog.FunctionBlocks.ArEventLogReadObjectID_0.Ident := EventLog.Data.Ident;
				EventLog.FunctionBlocks.ArEventLogReadObjectID_0.RecordID := EventLog.Event.RecordID;
				EventLog.FunctionBlocks.ArEventLogReadObjectID_0.Execute := TRUE;
			END_IF

		STEP_ERROR:        (*Do some error handling here.*)

			(* In case we try to delete a logger that is not there we will continue the execution from there,
			for other error ID's please see ArEventLog help *)
			IF EventLog.Data.StatusID = -1070586087 THEN
				EventLog.Data.StatusID := ERR_OK;
				EventLog.Data.Step := STEP_WAIT_FOR_INPUT;
			ELSE

			END_IF;
	END_CASE

    EventLog.FunctionBlocks.ArEventLogCreate_0;    EventLog.FunctionBlocks.ArEventLogDelete_0;    EventLog.FunctionBlocks.ArEventLogWrite_0;    EventLog.FunctionBlocks.ArEventLogGetIdent_0;    EventLog.FunctionBlocks.ArEventLogGetLatestRecordID_0;    EventLog.FunctionBlocks.ArEventLogGetPreviousRecordID_0;    EventLog.FunctionBlocks.ArEventLogReadAddData_0;    EventLog.FunctionBlocks.ArEventLogReadErrorNumber_0;    EventLog.FunctionBlocks.ArEventLogReadObjectID_0;    EventLog.FunctionBlocks.ArEventLogRead_0;END_PROGRAM

(*See ArEventLog help for the description of the event id format!*)

(*Gets severity from EventId (bits 31-30).*)
FUNCTION GetSeverity
	IF ArEventLogIsError(EventID := EventID) THEN
		GetSeverity := arEVENTLOG_SEVERITY_ERROR;
	ELSIF ArEventLogIsWarning(EventID := EventID) THEN
		GetSeverity := arEVENTLOG_SEVERITY_WARNING;
	ELSIF ArEventLogIsInformation(EventID := EventID) THEN
		GetSeverity := arEVENTLOG_SEVERITY_INFO;
	ELSIF ArEventLogIsSuccess(EventID := EventID) THEN
		GetSeverity := arEVENTLOG_SEVERITY_SUCCESS;
	END_IF
END_FUNCTION
(*Gets code from EventId (bits 15-0).*)
FUNCTION GetCode
	GetCode := DINT_TO_UINT(EventID);
END_FUNCTION

(*Gets facility from EventId (bits 27-16).*)
FUNCTION GetFacility
	GetFacility := DINT_TO_UINT(SHR(EventID, 16) AND 16#0FFF);
END_FUNCTION

PROGRAM _EXIT

	EventLog.FunctionBlocks.ArEventLogRead_0.Execute := FALSE;
	EventLog.FunctionBlocks.ArEventLogWrite_0.Execute := FALSE;
	EventLog.FunctionBlocks.ArEventLogGetLatestRecordID_0.Execute := FALSE;
	EventLog.FunctionBlocks.ArEventLogGetIdent_0.Execute := FALSE;

	EventLog.FunctionBlocks.ArEventLogRead_0();
	EventLog.FunctionBlocks.ArEventLogWrite_0();
	EventLog.FunctionBlocks.ArEventLogGetLatestRecordID_0();
	EventLog.FunctionBlocks.ArEventLogGetIdent_0();

END_PROGRAM
```

### Program Logical/HMI_Logic/Logic (IEC)

#### Main.st
```iecst
PROGRAM _INIT
	(* Insert code here *)

END_PROGRAM

PROGRAM _CYCLIC
	CASE gAssemblyModule.state.stateMachine.operationalState OF
		(*************************************************************************************************)
		(* RESETTING *)
		RESETTING:
			HMI_Assembly_State_String := 'RESETTING';

			(*************************************************************************************************)
			(* IDLE *)
		IDLE:
			HMI_Assembly_State_String := 'IDLE';
			(*************************************************************************************************)
			(* STARTING *)
		STARTING:
			HMI_Assembly_State_String := 'STARTING';
			(*************************************************************************************************)
			(* RUNNING *)
		RUNNING:
			HMI_Assembly_State_String := 'RUNNING';
			(*************************************************************************************************)
			(* PAUSING *)
		PAUSING:
			HMI_Assembly_State_String := 'PAUSING';
			(*************************************************************************************************)
			(* PAUSED *)
		PAUSED:
			HMI_Assembly_State_String := 'PAUSED';
			(*************************************************************************************************)
			(* SUSPENDING *)
		SUSPENDING:
			HMI_Assembly_State_String := 'SUSPENDING';
			(*************************************************************************************************)
			(* SUSPENDED *)
		SUSPENDED:
			HMI_Assembly_State_String := 'SUSPENDED';
			(*************************************************************************************************)
			(* UNSUSPENDING *)
		UNSUSPENDING:
			HMI_Assembly_State_String := 'UNSUSPENDING';
			(*************************************************************************************************)
			(* HOLDING *)
		HOLDING:
			HMI_Assembly_State_String := 'HOLDING';
			(*************************************************************************************************)
			(* HELD *)
		HELD:
			HMI_Assembly_State_String := 'HELD';
			(*************************************************************************************************)
			(* UNHOLDING *)
		UNHOLDING:
			HMI_Assembly_State_String := 'UNHOLDING';
			(*************************************************************************************************)
			(* COMPLETING *)
		COMPLETING:
			HMI_Assembly_State_String := 'COMPLETING';
			(*************************************************************************************************)
			(* COMPLETE *)
		COMPLETE:
			HMI_Assembly_State_String := 'COMPLETE';
			(*************************************************************************************************)
			(* STOPPING *)
		STOPPING:
			HMI_Assembly_State_String := 'STOPPING';
			(*************************************************************************************************)
			(* STOPPED *)
		STOPPED:
			HMI_Assembly_State_String := 'STOPPED';
			(*************************************************************************************************)
			(* ABORTING *)
		ABORTING:
			HMI_Assembly_State_String := 'ABORTING';
			(*************************************************************************************************)
			(* ABORTED *)
		ABORTED:
			HMI_Assembly_State_String := 'ABORTED';
			(*************************************************************************************************)
			(* CLEARING *)
		CLEARING:
			HMI_Assembly_State_String := 'CLEARING';
			(*************************************************************************************************)
			(* ELSE *)
		ELSE;
	END_CASE;

	CASE gSuperTrak.state.stateMachine.operationalState OF
		(*************************************************************************************************)
		(* RESETTING *)
		RESETTING:
			HMI_ST_State_String := 'RESETTING';

			(*************************************************************************************************)
			(* IDLE *)
		IDLE:
			HMI_ST_State_String := 'IDLE';
			(*************************************************************************************************)
			(* STARTING *)
		STARTING:
			HMI_ST_State_String := 'STARTING';
			(*************************************************************************************************)
			(* RUNNING *)
		RUNNING:
			HMI_ST_State_String := 'RUNNING';
			(*************************************************************************************************)
			(* PAUSING *)
		PAUSING:
			HMI_ST_State_String := 'PAUSING';
			(*************************************************************************************************)
			(* PAUSED *)
		PAUSED:
			HMI_ST_State_String := 'PAUSED';
			(*************************************************************************************************)
			(* SUSPENDING *)
		SUSPENDING:
			HMI_ST_State_String := 'SUSPENDING';
			(*************************************************************************************************)
			(* SUSPENDED *)
		SUSPENDED:
			HMI_ST_State_String := 'SUSPENDED';
			(*************************************************************************************************)
			(* UNSUSPENDING *)
		UNSUSPENDING:
			HMI_ST_State_String := 'UNSUSPENDING';
			(*************************************************************************************************)
			(* HOLDING *)
		HOLDING:
			HMI_ST_State_String := 'HOLDING';
			(*************************************************************************************************)
			(* HELD *)
		HELD:
			HMI_ST_State_String := 'HELD';
			(*************************************************************************************************)
			(* UNHOLDING *)
		UNHOLDING:
			HMI_ST_State_String := 'UNHOLDING';
			(*************************************************************************************************)
			(* COMPLETING *)
		COMPLETING:
			HMI_ST_State_String := 'COMPLETING';
			(*************************************************************************************************)
			(* COMPLETE *)
		COMPLETE:
			HMI_ST_State_String := 'COMPLETE';
			(*************************************************************************************************)
			(* STOPPING *)
		STOPPING:
			HMI_ST_State_String := 'STOPPING';
			(*************************************************************************************************)
			(* STOPPED *)
		STOPPED:
			HMI_ST_State_String := 'STOPPED';
			(*************************************************************************************************)
			(* ABORTING *)
		ABORTING:
			HMI_ST_State_String := 'ABORTING';
			(*************************************************************************************************)
			(* ABORTED *)
		ABORTED:
			HMI_ST_State_String := 'ABORTED';
			(*************************************************************************************************)
			(* CLEARING *)
		CLEARING:
			HMI_ST_State_String := 'CLEARING';
			(*************************************************************************************************)
			(* ELSE *)
		ELSE;
	END_CASE;

	IF HMI_Abort_System THEN
		gSuperTrak.state.stateMachine.stateTransition.abort 		:= TRUE;
		gAssemblyModule.state.stateMachine.stateTransition.abort 	:= TRUE;
	END_IF;

END_PROGRAM

PROGRAM _EXIT
	(* Insert code here *)

END_PROGRAM
```

Listed in the project but not available here: Logical/Opc.typ, Logical/Assembly_Module/MainControl/General_SM/StateMachine.st, Logical/Assembly_Module/MainControl/General_SM/Holding.st, Logical/Assembly_Module/MainControl/General_SM/Idle.st, Logical/Assembly_Module/MainControl/General_SM/Pausing.st, Logical/Assembly_Module/MainControl/General_SM/Starting.st, Logical/Assembly_Module/MainControl/General_SM/Suspending.st, Logical/Assembly_Module/MainControl/General_SM/Aborted.st, Logical/Assembly_Module/MainControl/General_SM/Complete.st, Logical/Assembly_Module/MainControl/General_SM/Aborting.st, Logical/Assembly_Module/MainControl/goHome_SM/goHome.st, Logical/Assembly_Module/MainControl/providePellet_SM/StateActions/providePellet_Aborting.st, Logical/Assembly_Module/MainControl/providePellet_SM/StateActions/providePellet_Aborted.st, Logical/Assembly_Module/MainControl/providePellet_SM/StateActions/providePellet_Stopping.st, Logical/Assembly_Module/MainControl/providePellet_SM/StateActions/providePellet_Stopped.st, Logical/Assembly_Module/MainControl/providePellet_SM/StateActions/providePellet_Resetting.st, Logical/Assembly_Module/MainControl/providePellet_SM/StateActions/providePellet_Held.st, Logical/Assembly_Module/MainControl/providePellet_SM/StateActions/providePellet_Pausing.st, Logical/Assembly_Module/MainControl/providePellet_SM/StateActions/providePellet_Running.st, Logical/Assembly_Module/MainControl/providePellet_SM/StateActions/providePellet_Paused.st, Logical/Assembly_Module/DisableBrake, Logical/Assembly_Module/Assembly_Global.var, Logical/Assembly_Module/MNG_Global.var, Logical/Assembly_Module/MNG_Interface/MNG_Interface.st, Logical/Assembly_Module/MNG_Interface/MNG_Interface.typ, Logical/Assembly_Module/MNG_Interface/MNG_Interface.var, Logical/Assembly_Module/MNG_Interface/MNG_COPY_OUTPUTS_INTO_MSG.st, Logical/SuperTrak_Module/StateMachine_SuperTrak/Main.st, Logical/SuperTrak_Module/StateMachine_SuperTrak/StateActions/Resetting.st, Logical/SuperTrak_Module/StateMachine_SuperTrak/StateActions/Idle.st, Logical/SuperTrak_Module/StateMachine_SuperTrak/StateActions/Starting.st, Logical/SuperTrak_Module/StateMachine_SuperTrak/StateActions/Pausing.st, Logical/SuperTrak_Module/StateMachine_SuperTrak/StateActions/Suspended.st, Logical/SuperTrak_Module/StateMachine_SuperTrak/StateActions/Completing.st, Logical/SuperTrak_Module/StateMachine_SuperTrak/checkParking/checkParking.st, Logical/SuperTrak_Module/StateMachine_SuperTrak/checkParking/StateActions/checkParking_Aborted.st, Logical/SuperTrak_Module/StateMachine_SuperTrak/checkParking/StateActions/checkParking_Stopping.st, Logical/SuperTrak_Module/StateMachine_SuperTrak/checkParking/StateActions/checkParking_Clearing.st, Logical/SuperTrak_Module/StateMachine_SuperTrak/checkParking/StateActions/checkParking_Starting.st, Logical/SuperTrak_Module/StateMachine_SuperTrak/checkParking/StateActions/checkParking_Completing.st, Logical/SuperTrak_Module/StateMachine_SuperTrak/checkParking/StateActions/checkParking_Complete.st, Logical/SuperTrak_Module/StateMachine_SuperTrak/checkParking/StateActions/checkParking_Unholding.st, Logical/SuperTrak_Module/StateMachine_SuperTrak/checkParking/StateActions/checkParking_Suspending.st, Logical/SuperTrak_Module/StateMachine_SuperTrak/checkParking/StateActions/checkParking_Unsuspending.st, Logical/SuperTrak_Module/StateMachine_SuperTrak/checkParking/StateActions/checkParking_Pausing.st, Logical/SuperTrak_Module/StateMachine_SuperTrak/Outfeed/StateActions/Outfeed_Stopping.st, Logical/SuperTrak_Module/StateMachine_SuperTrak/Outfeed/StateActions/Outfeed_Idle.st, Logical/SuperTrak_Module/StateMachine_SuperTrak/Outfeed/StateActions/Outfeed_Resetting.st, Logical/SuperTrak_Module/StateMachine_SuperTrak/Outfeed/StateActions/Outfeed_Held.st, Logical/SuperTrak_Module/StateMachine_SuperTrak/Outfeed/StateActions/Outfeed_Unholding.st, Logical/SuperTrak_Module/StateMachine_SuperTrak/Outfeed/StateActions/Outfeed_Suspending.st, Logical/SuperTrak_Module/StateMachine_SuperTrak/Outfeed/StateActions/Outfeed_Pausing.st, Logical/SuperTrak_Module/StateMachine_SuperTrak/Outfeed/StateActions/Outfeed_Paused.st, Logical/SuperTrak_Module/StateMachine_SuperTrak/QACheck/StateActions/QACheck_Stopping.st, Logical/SuperTrak_Module/StateMachine_SuperTrak/QACheck/StateActions/QACheck_Stopped.st, Logical/SuperTrak_Module/StateMachine_SuperTrak/QACheck/StateActions/QACheck_Resetting.st, Logical/SuperTrak_Module/StateMachine_SuperTrak/QACheck/StateActions/QACheck_Held.st, Logical/SuperTrak_Module/StateMachine_SuperTrak/QACheck/StateActions/QACheck_Unholding.st, Logical/SuperTrak_Module/StateMachine_SuperTrak/QACheck/StateActions/QACheck_Suspending.st, Logical/SuperTrak_Module/StateMachine_SuperTrak/QACheck/StateActions/QACheck_Suspended.st, Logical/SuperTrak_Module/StateMachine_SuperTrak/QACheck/StateActions/QACheck_Unsuspending.st, Logical/SuperTrak_Module/StateMachine_SuperTrak/QACheck/StateActions/QACheck_Pausing.st, Logical/SuperTrak_Module/StateMachine_SuperTrak/QACheck/StateActions/QACheck_Paused.st, Logical/SuperTrak_Module/StateMachine_SuperTrak/QACheck/StateActions/QACheck_Holding.st, Logical/Events_handling/AlarmHandling/Error_Handling/ServiceStations.st, Logical/Events_handling/AlarmHandling/Event_Handling/ErrorSum.st, Logical/Events_handling/AlarmHandling/Event_Handling/StateInfo.st, Logical/Events_handling/AlarmHandling/Events_Definition/Common_Events.st, Logical/Global.typ
